# B&R Automation Studio project 8238 (part 4)

```iecst
(*** RAIL DEST MAPPING FOR RAIL DESTINATIONS ***)

DEST_SIZE := rail_destination_1;
DEST_RAIL := 0;
DEST_NUM := 0;
IF DEST_SIZE > 0 THEN
	FOR DEST_INDEX := 1 TO DEST_SIZE DO
		CASE DEST_INDEX OF
		1:	DEST_RAIL := rail_destination_2; DEST_NUM := rail_destination_3;
		2:	DEST_RAIL := rail_destination_4; DEST_NUM := rail_destination_5;
		3:	DEST_RAIL := rail_destination_6; DEST_NUM := rail_destination_7;
		4:	DEST_RAIL := rail_destination_8; DEST_NUM := rail_destination_9;
		5:	DEST_RAIL := rail_destination_10; DEST_NUM := rail_destination_11;
		6:	DEST_RAIL := rail_destination_12; DEST_NUM := rail_destination_13;
		7:	DEST_RAIL := rail_destination_14; DEST_NUM := rail_destination_15;
		8:	DEST_RAIL := rail_destination_16; DEST_NUM := rail_destination_17;
		9:	DEST_RAIL := rail_destination_18; DEST_NUM := rail_destination_19;
		10:	DEST_RAIL := rail_destination_20; DEST_NUM := rail_destination_21;
		11:	DEST_RAIL := rail_destination_22; DEST_NUM := rail_destination_23;
		12:	DEST_RAIL := rail_destination_24; DEST_NUM := rail_destination_25;
		13:	DEST_RAIL := rail_destination_26; DEST_NUM := rail_destination_27;
		14:	DEST_RAIL := rail_destination_28; DEST_NUM := rail_destination_29;
		15:	DEST_RAIL := rail_destination_30; DEST_NUM := rail_destination_31;
		16:	DEST_RAIL := rail_destination_32; DEST_NUM := rail_destination_33;
		17:	DEST_RAIL := rail_destination_34; DEST_NUM := rail_destination_35;
		18:	DEST_RAIL := rail_destination_36; DEST_NUM := rail_destination_37;
		19:	DEST_RAIL := rail_destination_38; DEST_NUM := rail_destination_39;
		20:	DEST_RAIL := rail_destination_40; DEST_NUM := rail_destination_41;
		21:	DEST_RAIL := rail_destination_42; DEST_NUM := rail_destination_43;
		22:	DEST_RAIL := rail_destination_44; DEST_NUM := rail_destination_45;
		23:	DEST_RAIL := rail_destination_46; DEST_NUM := rail_destination_47;
		24:	DEST_RAIL := rail_destination_48; DEST_NUM := rail_destination_49;
		25:	DEST_RAIL := rail_destination_50; DEST_NUM := rail_destination_51;
		26:	DEST_RAIL := rail_destination_52; DEST_NUM := rail_destination_53;
		27:	DEST_RAIL := rail_destination_54; DEST_NUM := rail_destination_55;
		28:	DEST_RAIL := rail_destination_56; DEST_NUM := rail_destination_57;
		29:	DEST_RAIL := rail_destination_58; DEST_NUM := rail_destination_59;
		30:	DEST_RAIL := rail_destination_60; DEST_NUM := rail_destination_61;
		31:	DEST_RAIL := rail_destination_62; DEST_NUM := rail_destination_63;
		32:	DEST_RAIL := rail_destination_64; DEST_NUM := rail_destination_65;
		33:	DEST_RAIL := rail_destination_66; DEST_NUM := rail_destination_67;
		34:	DEST_RAIL := rail_destination_68; DEST_NUM := rail_destination_69;
		35:	DEST_RAIL := rail_destination_70; DEST_NUM := rail_destination_71;
		36:	DEST_RAIL := rail_destination_72; DEST_NUM := rail_destination_73;
		37:	DEST_RAIL := rail_destination_74; DEST_NUM := rail_destination_75;
		38:	DEST_RAIL := rail_destination_76; DEST_NUM := rail_destination_77;
		39:	DEST_RAIL := rail_destination_78; DEST_NUM := rail_destination_79;
		40:	DEST_RAIL := rail_destination_80; DEST_NUM := rail_destination_81;
		41:	DEST_RAIL := rail_destination_82; DEST_NUM := rail_destination_83;
		42:	DEST_RAIL := rail_destination_84; DEST_NUM := rail_destination_85;
		43:	DEST_RAIL := rail_destination_86; DEST_NUM := rail_destination_87;
		44:	DEST_RAIL := rail_destination_88; DEST_NUM := rail_destination_89;
		45:	DEST_RAIL := rail_destination_90; DEST_NUM := rail_destination_91;
		46:	DEST_RAIL := rail_destination_92; DEST_NUM := rail_destination_93;
		47:	DEST_RAIL := rail_destination_94; DEST_NUM := rail_destination_95;
		48:	DEST_RAIL := rail_destination_96; DEST_NUM := rail_destination_97;
		49:	DEST_RAIL := rail_destination_98; DEST_NUM := rail_destination_99;
		50:	DEST_RAIL := rail_destination_100; DEST_NUM := rail_destination_101;
		END_CASE;
		CASE DEST_RAIL OF
		1:	r1.destination := DEST_NUM;
		2:	r2.destination := DEST_NUM;
		3:	r3.destination := DEST_NUM;
		4:	r4.destination := DEST_NUM;
		5:	r5.destination := DEST_NUM;
		6:	r6.destination := DEST_NUM;
		7:	r7.destination := DEST_NUM;
		8:	r8.destination := DEST_NUM;
		9:	r9.destination := DEST_NUM;
		10:	r10.destination := DEST_NUM;
		11:	r11.destination := DEST_NUM;
		12:	r12.destination := DEST_NUM;
		13:	r13.destination := DEST_NUM;
		14:	r14.destination := DEST_NUM;
		15:	r15.destination := DEST_NUM;
		16:	r16.destination := DEST_NUM;
		17:	r17.destination := DEST_NUM;
		18:	r18.destination := DEST_NUM;
		19:	r19.destination := DEST_NUM;
		20:	r20.destination := DEST_NUM;
		21:	r21.destination := DEST_NUM;
		22:	r22.destination := DEST_NUM;
		23:	r23.destination := DEST_NUM;
		24:	r24.destination := DEST_NUM;
		25:	r25.destination := DEST_NUM;
		26:	r26.destination := DEST_NUM;
		27:	r27.destination := DEST_NUM;
		28:	r28.destination := DEST_NUM;
		29:	r29.destination := DEST_NUM;
		30:	r30.destination := DEST_NUM;
		31:	r31.destination := DEST_NUM;
		32:	r32.destination := DEST_NUM;
		33:	r33.destination := DEST_NUM;
		34:	r34.destination := DEST_NUM;
		35:	r35.destination := DEST_NUM;
		36:	r36.destination := DEST_NUM;
		37:	r37.destination := DEST_NUM;
		38:	r38.destination := DEST_NUM;
		39:	r39.destination := DEST_NUM;
		40:	r40.destination := DEST_NUM;
		41:	r41.destination := DEST_NUM;
		42:	r42.destination := DEST_NUM;
		43:	r43.destination := DEST_NUM;
		44:	r44.destination := DEST_NUM;
		45:	r45.destination := DEST_NUM;
		46:	r46.destination := DEST_NUM;
		47:	r47.destination := DEST_NUM;
		48:	r48.destination := DEST_NUM;
		49:	r49.destination := DEST_NUM;
		50:	r50.destination := DEST_NUM;
		51:	r51.destination := DEST_NUM;
		52:	r52.destination := DEST_NUM;
		53:	r53.destination := DEST_NUM;
		54:	r54.destination := DEST_NUM;
		55:	r55.destination := DEST_NUM;
		56:	r56.destination := DEST_NUM;
		57:	r57.destination := DEST_NUM;
		58:	r58.destination := DEST_NUM;
		59:	r59.destination := DEST_NUM;
		60:	r60.destination := DEST_NUM;
		61:	r61.destination := DEST_NUM;
		62:	r62.destination := DEST_NUM;
		63:	r63.destination := DEST_NUM;
		64:	r64.destination := DEST_NUM;
		65:	r65.destination := DEST_NUM;
		66:	r66.destination := DEST_NUM;
		67:	r67.destination := DEST_NUM;
		68:	r68.destination := DEST_NUM;
		69:	r69.destination := DEST_NUM;
		70:	r70.destination := DEST_NUM;
		71:	r71.destination := DEST_NUM;
		72:	r72.destination := DEST_NUM;
		73:	r73.destination := DEST_NUM;
		74:	r74.destination := DEST_NUM;
		END_CASE;
	END_FOR;
END_IF;
rail_destination_1 := 0;
rail_destination_2 := 0;
rail_destination_3 := 0;
rail_destination_4 := 0;
rail_destination_5 := 0;
rail_destination_6 := 0;
rail_destination_7 := 0;
rail_destination_8 := 0;
rail_destination_9 := 0;
rail_destination_10 := 0;
rail_destination_11 := 0;
rail_destination_12 := 0;
rail_destination_13 := 0;
rail_destination_14 := 0;
rail_destination_15 := 0;
rail_destination_16 := 0;
rail_destination_17 := 0;
rail_destination_18 := 0;
rail_destination_19 := 0;
rail_destination_20 := 0;
rail_destination_21 := 0;
rail_destination_22 := 0;
rail_destination_23 := 0;
rail_destination_24 := 0;
rail_destination_25 := 0;
rail_destination_26 := 0;
rail_destination_27 := 0;
rail_destination_28 := 0;
rail_destination_29 := 0;
rail_destination_30 := 0;
rail_destination_31 := 0;
rail_destination_32 := 0;
rail_destination_33 := 0;
rail_destination_34 := 0;
rail_destination_35 := 0;
rail_destination_36 := 0;
rail_destination_37 := 0;
rail_destination_38 := 0;
rail_destination_39 := 0;
rail_destination_40 := 0;
rail_destination_41 := 0;
rail_destination_42 := 0;
rail_destination_43 := 0;
rail_destination_44 := 0;
rail_destination_45 := 0;
rail_destination_46 := 0;
rail_destination_47 := 0;
rail_destination_48 := 0;
rail_destination_49 := 0;
rail_destination_50 := 0;
rail_destination_51 := 0;
rail_destination_52 := 0;
rail_destination_53 := 0;
rail_destination_54 := 0;
rail_destination_55 := 0;
rail_destination_56 := 0;
rail_destination_57 := 0;
rail_destination_58 := 0;
rail_destination_59 := 0;
rail_destination_60 := 0;
rail_destination_61 := 0;
rail_destination_62 := 0;
rail_destination_63 := 0;
rail_destination_64 := 0;
rail_destination_65 := 0;
rail_destination_66 := 0;
rail_destination_67 := 0;
rail_destination_68 := 0;
rail_destination_69 := 0;
rail_destination_70 := 0;
rail_destination_71 := 0;
rail_destination_72 := 0;
rail_destination_73 := 0;
rail_destination_74 := 0;
rail_destination_75 := 0;
rail_destination_76 := 0;
rail_destination_77 := 0;
rail_destination_78 := 0;
rail_destination_79 := 0;
rail_destination_80 := 0;
rail_destination_81 := 0;
rail_destination_82 := 0;
rail_destination_83 := 0;
rail_destination_84 := 0;
rail_destination_85 := 0;
rail_destination_86 := 0;
rail_destination_87 := 0;
rail_destination_88 := 0;
rail_destination_89 := 0;
rail_destination_90 := 0;
rail_destination_91 := 0;
rail_destination_92 := 0;
rail_destination_93 := 0;
rail_destination_94 := 0;
rail_destination_95 := 0;
rail_destination_96 := 0;
rail_destination_97 := 0;
rail_destination_98 := 0;
rail_destination_99 := 0;
rail_destination_100 := 0;
rail_destination_101 := 0;

(*** RESET CLEARING DEST, FIRE, AND GOING_TO ***)

(*** Rail 1 ***)
IF r1.reset THEN
	r1.fire := 0;
	IF r1.destination = 61 THEN
		r61.going_to := 0;
	END_IF;
	r1.destination := 0;
END_IF;

(*** Rail 2 ***)
IF r2.reset THEN
	r2.fire := 0;
	IF r2.destination = 61 THEN
		r61.going_to := 0;
	END_IF;
	r2.destination := 0;
END_IF;

(*** Rail 3 ***)
IF r3.reset THEN
	r3.fire := 0;
	IF r3.destination = 61 THEN
		r61.going_to := 0;
	END_IF;
	r3.destination := 0;
END_IF;

(*** Rail 4 ***)
IF r4.reset THEN
	r4.fire := 0;
	IF r4.destination = 61 THEN
		r61.going_to := 0;
	END_IF;
	r4.destination := 0;
END_IF;

(*** Rail 5 ***)
IF r5.reset THEN
	r5.fire := 0;
	IF r5.destination = 61 THEN
		r61.going_to := 0;
	END_IF;
	r5.destination := 0;
END_IF;

(*** Rail 6 ***)
IF r6.reset THEN
	r6.fire := 0;
	IF r6.destination = 61 THEN
		r61.going_to := 0;
	END_IF;
	r6.destination := 0;
END_IF;

(*** Rail 7 ***)
IF r7.reset THEN
	r7.fire := 0;
	IF r7.destination = 61 THEN
		r61.going_to := 0;
	END_IF;
	r7.destination := 0;
END_IF;

(*** Rail 8 ***)
IF r8.reset THEN
	r8.fire := 0;
	IF r8.destination = 61 THEN
		r61.going_to := 0;
	END_IF;
	r8.destination := 0;
END_IF;

(*** Rail 9 ***)
IF r9.reset THEN
	r9.fire := 0;
	IF r9.destination = 61 THEN
		r61.going_to := 0;
	END_IF;
	r9.destination := 0;
END_IF;

(*** Rail 10 ***)
IF r10.reset THEN
	r10.fire := 0;
	IF r10.destination = 61 THEN
		r61.going_to := 0;
	END_IF;
	r10.destination := 0;
END_IF;

(*** Rail 11 ***)
IF r11.reset THEN
	r11.fire := 0;
	IF r11.destination = 61 THEN
		r61.going_to := 0;
	END_IF;
	r11.destination := 0;
END_IF;

(*** Rail 12 ***)
IF r12.reset THEN
	r12.fire := 0;
	IF r12.destination = 63 THEN
		r63.going_to := 0;
	END_IF;
	r12.destination := 0;
END_IF;

(*** Rail 13 ***)
IF r13.reset THEN
	r13.fire := 0;
	IF r13.destination = 63 THEN
		r63.going_to := 0;
	END_IF;
	r13.destination := 0;
END_IF;

(*** Rail 14 ***)
IF r14.reset THEN
	r14.fire := 0;
	IF r14.destination = 63 THEN
		r63.going_to := 0;
	END_IF;
	r14.destination := 0;
END_IF;

(*** Rail 15 ***)
IF r15.reset THEN
	r15.fire := 0;
	IF r15.destination = 63 THEN
		r63.going_to := 0;
	END_IF;
	r15.destination := 0;
END_IF;

(*** Rail 16 ***)
IF r16.reset THEN
	r16.fire := 0;
	IF r16.destination = 63 THEN
		r63.going_to := 0;
	END_IF;
	r16.destination := 0;
END_IF;

(*** Rail 17 ***)
IF r17.reset THEN
	r17.fire := 0;
	IF r17.destination = 63 THEN
		r63.going_to := 0;
	END_IF;
	r17.destination := 0;
END_IF;

(*** Rail 18 ***)
IF r18.reset THEN
	r18.fire := 0;
	IF r18.destination = 63 THEN
		r63.going_to := 0;
	END_IF;
	r18.destination := 0;
END_IF;

(*** Rail 19 ***)
IF r19.reset THEN
	r19.fire := 0;
	IF r19.destination = 63 THEN
		r63.going_to := 0;
	END_IF;
	r19.destination := 0;
END_IF;

(*** Rail 20 ***)
IF r20.reset THEN
	r20.fire := 0;
	IF r20.destination = 63 THEN
		r63.going_to := 0;
	END_IF;
	r20.destination := 0;
END_IF;

(*** Rail 21 ***)
IF r21.reset THEN
	r21.fire := 0;
	IF r21.destination = 63 THEN
		r63.going_to := 0;
	END_IF;
	r21.destination := 0;
END_IF;

(*** Rail 22 ***)
IF r22.reset THEN
	r22.fire := 0;
	IF r22.destination = 63 THEN
		r63.going_to := 0;
	END_IF;
	r22.destination := 0;
END_IF;

(*** Rail 23 ***)
IF r23.reset THEN
	r23.fire := 0;
	IF r23.destination = 63 THEN
		r63.going_to := 0;
	END_IF;
	r23.destination := 0;
END_IF;

(*** Rail 24 ***)
IF r24.reset THEN
	r24.fire := 0;
	IF r24.destination = 63 THEN
		r63.going_to := 0;
	END_IF;
	r24.destination := 0;
END_IF;

(*** Rail 25 ***)
IF r25.reset THEN
	r25.fire := 0;
	IF r25.destination = 63 THEN
		r63.going_to := 0;
	END_IF;
	r25.destination := 0;
END_IF;

(*** Rail 26 ***)
IF r26.reset THEN
	r26.fire := 0;
	IF r26.destination = 63 THEN
		r63.going_to := 0;
	END_IF;
	r26.destination := 0;
END_IF;

(*** Rail 27 ***)
IF r27.reset THEN
	r27.fire := 0;
	IF r27.destination = 63 THEN
		r63.going_to := 0;
	END_IF;
	r27.destination := 0;
END_IF;

(*** Rail 28 ***)
IF r28.reset THEN
	r28.fire := 0;
	IF r28.destination = 63 THEN
		r63.going_to := 0;
	END_IF;
	r28.destination := 0;
END_IF;

(*** Rail 29 ***)
IF r29.reset THEN
	r29.fire := 0;
	IF r29.destination = 63 THEN
		r63.going_to := 0;
	END_IF;
	r29.destination := 0;
END_IF;

(*** Rail 30 ***)
IF r30.reset THEN
	r30.fire := 0;
	IF r30.destination = 63 THEN
		r63.going_to := 0;
	END_IF;
	r30.destination := 0;
END_IF;

(*** Rail 31 ***)
IF r31.reset THEN
	r31.fire := 0;
	IF r31.destination = 63 THEN
		r63.going_to := 0;
	END_IF;
	r31.destination := 0;
END_IF;

(*** Rail 32 ***)
IF r32.reset THEN
	r32.fire := 0;
	IF r32.destination = 63 THEN
		r63.going_to := 0;
	END_IF;
	r32.destination := 0;
END_IF;

(*** Rail 33 ***)
IF r33.reset THEN
	r33.fire := 0;
	IF r33.destination = 63 THEN
		r63.going_to := 0;
	END_IF;
	r33.destination := 0;
END_IF;

(*** Rail 34 ***)
IF r34.reset THEN
	r34.fire := 0;
	IF r34.destination = 63 THEN
		r63.going_to := 0;
	END_IF;
	r34.destination := 0;
END_IF;

(*** Rail 35 ***)
IF r35.reset THEN
	r35.fire := 0;
	IF r35.destination = 63 THEN
		r63.going_to := 0;
	END_IF;
	r35.destination := 0;
END_IF;

(*** Rail 36 ***)
IF r36.reset THEN
	r36.fire := 0;
	IF r36.destination = 63 THEN
		r63.going_to := 0;
	END_IF;
	r36.destination := 0;
END_IF;

(*** Rail 37 ***)
IF r37.reset THEN
	r37.fire := 0;
	IF r37.destination = 66 THEN
		r66.going_to := 0;
	END_IF;
	r37.destination := 0;
END_IF;

(*** Rail 38 ***)
IF r38.reset THEN
	r38.fire := 0;
	IF r38.destination = 66 THEN
		r66.going_to := 0;
	END_IF;
	r38.destination := 0;
END_IF;

(*** Rail 39 ***)
IF r39.reset THEN
	r39.fire := 0;
	IF r39.destination = 66 THEN
		r66.going_to := 0;
	END_IF;
	r39.destination := 0;
END_IF;

(*** Rail 40 ***)
IF r40.reset THEN
	r40.fire := 0;
	IF r40.destination = 66 THEN
		r66.going_to := 0;
	END_IF;
	r40.destination := 0;
END_IF;

(*** Rail 41 ***)
IF r41.reset THEN
	r41.fire := 0;
	IF r41.destination = 66 THEN
		r66.going_to := 0;
	END_IF;
	r41.destination := 0;
END_IF;

(*** Rail 42 ***)
IF r42.reset THEN
	r42.fire := 0;
	IF r42.destination = 66 THEN
		r66.going_to := 0;
	END_IF;
	r42.destination := 0;
END_IF;

(*** Rail 43 ***)
IF r43.reset THEN
	r43.fire := 0;
	IF r43.destination = 65 THEN
		r65.going_to := 0;
	END_IF;
	r43.destination := 0;
END_IF;

(*** Rail 44 ***)
IF r44.reset THEN
	r44.fire := 0;
	IF r44.destination = 65 THEN
		r65.going_to := 0;
	END_IF;
	r44.destination := 0;
END_IF;

(*** Rail 45 ***)
IF r45.reset THEN
	r45.fire := 0;
	IF r45.destination = 65 THEN
		r65.going_to := 0;
	END_IF;
	r45.destination := 0;
END_IF;

(*** Rail 46 ***)
IF r46.reset THEN
	r46.fire := 0;
	IF r46.destination = 65 THEN
		r65.going_to := 0;
	END_IF;
	r46.destination := 0;
END_IF;

(*** Rail 47 ***)
IF r47.reset THEN
	r47.fire := 0;
	IF r47.destination = 65 THEN
		r65.going_to := 0;
	END_IF;
	r47.destination := 0;
END_IF;

(*** Rail 48 ***)
IF r48.reset THEN
	r48.fire := 0;
	IF r48.destination = 65 THEN
		r65.going_to := 0;
	END_IF;
	r48.destination := 0;
END_IF;

(*** Rail 49 ***)
IF r49.reset THEN
	r49.fire := 0;
	IF r49.destination = 69 THEN
		r69.going_to := 0;
	END_IF;
	r49.destination := 0;
END_IF;

(*** Rail 50 ***)
IF r50.reset THEN
	r50.fire := 0;
	IF r50.destination = 69 THEN
		r69.going_to := 0;
	END_IF;
	r50.destination := 0;
END_IF;

(*** Rail 51 ***)
IF r51.reset THEN
	r51.fire := 0;
	IF r51.destination = 69 THEN
		r69.going_to := 0;
	END_IF;
	r51.destination := 0;
END_IF;

(*** Rail 52 ***)
IF r52.reset THEN
	r52.fire := 0;
	IF r52.destination = 69 THEN
		r69.going_to := 0;
	END_IF;
	r52.destination := 0;
END_IF;

(*** Rail 53 ***)
IF r53.reset THEN
	r53.fire := 0;
	IF r53.destination = 69 THEN
		r69.going_to := 0;
	END_IF;
	r53.destination := 0;
END_IF;

(*** Rail 54 ***)
IF r54.reset THEN
	r54.fire := 0;
	IF r54.destination = 69 THEN
		r69.going_to := 0;
	END_IF;
	r54.destination := 0;
END_IF;

(*** Rail 55 ***)
IF r55.reset THEN
	r55.fire := 0;
	IF r55.destination = 68 THEN
		r68.going_to := 0;
	END_IF;
	r55.destination := 0;
END_IF;

(*** Rail 56 ***)
IF r56.reset THEN
	r56.fire := 0;
	IF r56.destination = 68 THEN
		r68.going_to := 0;
	END_IF;
	r56.destination := 0;
END_IF;

(*** Rail 57 ***)
IF r57.reset THEN
	r57.fire := 0;
	IF r57.destination = 68 THEN
		r68.going_to := 0;
	END_IF;
	r57.destination := 0;
END_IF;

(*** Rail 58 ***)
IF r58.reset THEN
	r58.fire := 0;
	IF r58.destination = 68 THEN
		r68.going_to := 0;
	END_IF;
	r58.destination := 0;
END_IF;

(*** Rail 59 ***)
IF r59.reset THEN
	r59.fire := 0;
	IF r59.destination = 68 THEN
		r68.going_to := 0;
	END_IF;
	r59.destination := 0;
END_IF;

(*** Rail 60 ***)
IF r60.reset THEN
	r60.fire := 0;
	IF r60.destination = 68 THEN
		r68.going_to := 0;
	END_IF;
	r60.destination := 0;
END_IF;

(*** Rail 61 ***)
IF r61.reset THEN
	r61.fire := 0;
	r61.destination := 0;
END_IF;

(*** Rail 62 ***)
IF r62.reset THEN
	r62.fire := 0;
	r62.destination := 0;
END_IF;

(*** Rail 63 ***)
IF r63.reset THEN
	r63.fire := 0;
	r63.destination := 0;
END_IF;

(*** Rail 64 ***)
IF r64.reset THEN
	r64.fire := 0;
	r64.destination := 0;
END_IF;

(*** Rail 65 ***)
IF r65.reset THEN
	r65.fire := 0;
	r65.destination := 0;
END_IF;

(*** Rail 66 ***)
IF r66.reset THEN
	r66.fire := 0;
	r66.destination := 0;
END_IF;

(*** Rail 67 ***)
IF r67.reset THEN
	r67.fire := 0;
	r67.destination := 0;
END_IF;

(*** Rail 68 ***)
IF r68.reset THEN
	r68.fire := 0;
	r68.destination := 0;
END_IF;

(*** Rail 69 ***)
IF r69.reset THEN
	r69.fire := 0;
	r69.destination := 0;
END_IF;

(*** Rail 70 ***)
IF r70.reset THEN
	r70.fire := 0;
	r70.destination := 0;
END_IF;

(*** Rail 71 ***)
IF r71.reset THEN
	r71.fire := 0;
	r71.destination := 0;
END_IF;

(*** Rail 72 ***)
IF r72.reset THEN
	r72.fire := 0;
	r72.destination := 0;
END_IF;

(*** Rail 73 ***)
IF r73.reset THEN
	r73.fire := 0;
	r73.destination := 0;
END_IF;

(*** Rail 74 ***)
IF r74.reset THEN
	r74.fire := 0;
	r74.destination := 0;
END_IF;

(*** Conveyor Stop Signals ***)

conveyor_stop_1 := conveyor_stop_word_1.0;
conveyor_stop_2 := conveyor_stop_word_1.1;
conveyor_stop_3 := conveyor_stop_word_1.2;
conveyor_stop_4 := conveyor_stop_word_1.3;

END_PROGRAM
```

### Program Logical/LIFTS (IEC, version 1.00.1)

#### LIFTS.st
```iecst
(********************************************************************
 * Program: lifts
 * File: lifts.st
 ********************************************************************)
PROGRAM _CYCLIC
END_PROGRAM
```

#### Variables.var - not listed in the package file held
```iecst
VAR
	slant_timeout : BOOL;
	test_bit_a : BOOL;
	test_bit_b : BOOL;
END_VAR
```

#### Cyclic.ld - not listed in the package file held
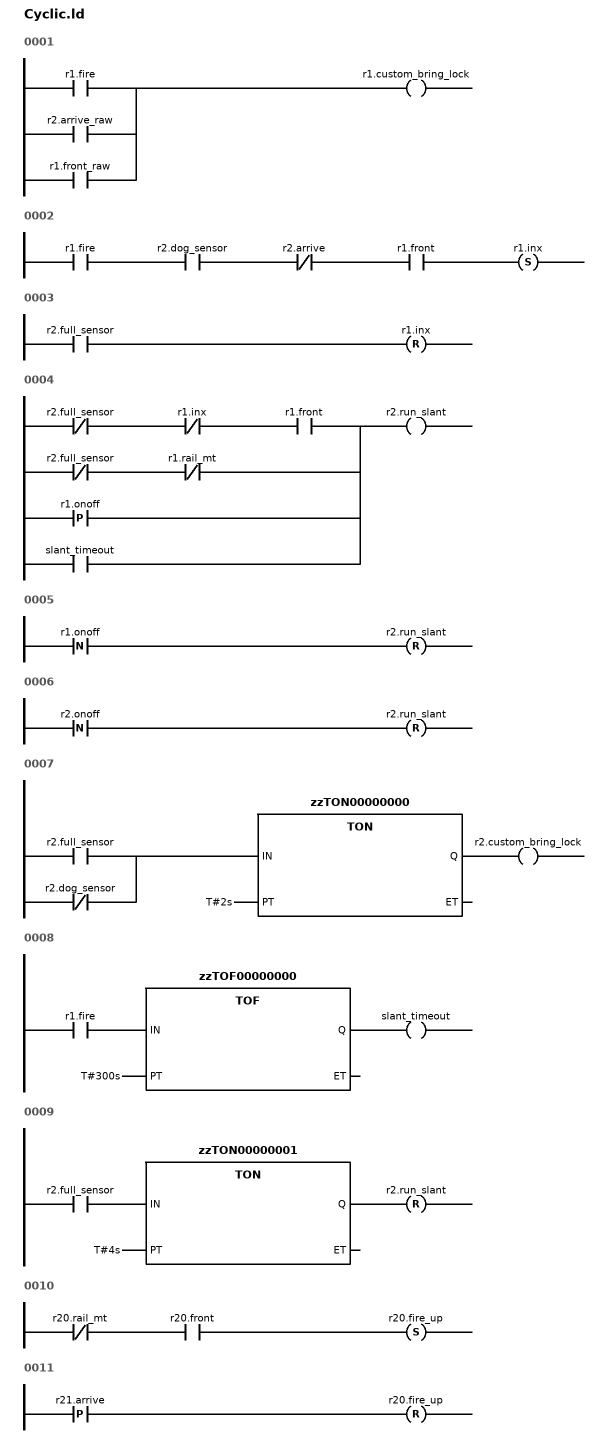
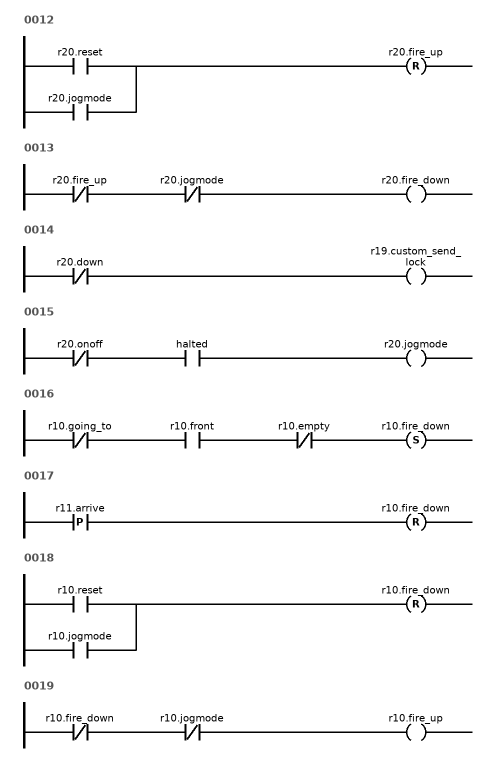
Ladder, written as Structured Text:
```iecst
PROGRAM _CYCLIC
VAR
    _e1 : R_TRIG;
    _e2 : F_TRIG;
    _e3 : F_TRIG;
    _e4 : R_TRIG;
    _e5 : R_TRIG;
END_VAR
(* Network 1 *)
r1.custom_bring_lock := r1.fire OR r2.arrive_raw OR r1.front_raw;

(* Network 2 *)
IF r1.fire AND r2.dog_sensor AND NOT r2.arrive AND r1.front THEN r1.inx := TRUE; END_IF;

(* Network 3 *)
IF r2.full_sensor THEN r1.inx := FALSE; END_IF;

(* Network 4 *)
_e1(CLK := r1.onoff);
r2.run_slant := (NOT r2.full_sensor AND ((NOT r1.inx AND r1.front) OR NOT r1.rail_mt)) OR _e1.Q OR slant_timeout;

(* Network 5 *)
_e2(CLK := r1.onoff);
IF _e2.Q THEN r2.run_slant := FALSE; END_IF;

(* Network 6 *)
_e3(CLK := r2.onoff);
IF _e3.Q THEN r2.run_slant := FALSE; END_IF;

(* Network 7 *)
zzTON00000000(IN := r2.full_sensor OR NOT r2.dog_sensor, PT := T#2s);
r2.custom_bring_lock := zzTON00000000.Q;

(* Network 8 *)
zzTOF00000000(IN := r1.fire, PT := T#300s);
slant_timeout := zzTOF00000000.Q;

(* Network 9 *)
zzTON00000001(IN := r2.full_sensor, PT := T#4s);
IF zzTON00000001.Q THEN r2.run_slant := FALSE; END_IF;

(* Network 10 *)
IF NOT r20.rail_mt AND r20.front THEN r20.fire_up := TRUE; END_IF;

(* Network 11 *)
_e4(CLK := r21.arrive);
IF _e4.Q THEN r20.fire_up := FALSE; END_IF;

(* Network 12 *)
IF r20.reset OR r20.jogmode THEN r20.fire_up := FALSE; END_IF;

(* Network 13 *)
r20.fire_down := NOT r20.fire_up AND NOT r20.jogmode;

(* Network 14 *)
r19.custom_send_lock := NOT r20.down;

(* Network 15 *)
r20.jogmode := NOT r20.onoff AND halted;

(* Network 16 *)
IF NOT r10.going_to AND r10.front AND NOT r10.empty THEN r10.fire_down := TRUE; END_IF;

(* Network 17 *)
_e5(CLK := r11.arrive);
IF _e5.Q THEN r10.fire_down := FALSE; END_IF;

(* Network 18 *)
IF r10.reset OR r10.jogmode THEN r10.fire_down := FALSE; END_IF;

(* Network 19 *)
r10.fire_up := NOT r10.fire_down AND NOT r10.jogmode;
END_PROGRAM
```

### Program Logical/RAIL_SUB (IEC, version 1.00.1) - RAIL_SUB

#### RAIL_SUB.st
```iecst
(********************************************************************
 * Program: st_rails
 * File: st_rails.st
 ********************************************************************)
PROGRAM _CYCLIC
(***	RAILS	***)
(*
  This section maps the plc state of io_ok and manages fire bits
*)

	(***	Rail: 1	***)
	IF r1.fire_ns THEN r1.destination := 0; END_IF;
	IF r1.destination = 61 THEN
		IF NOT(r61.going_to) AND NOT(r1.reset) AND NOT(r61.insert_reset) THEN
			r61.going_to := TRUE;
			r1.fire := TRUE;
		END_IF;

		IF r1.fire AND r61.insert_reset THEN
			r1.fire := FALSE;
		END_IF;
	END_IF;

	(***	Rail: 2	***)
	IF r2.fire_ns THEN r2.destination := 0; END_IF;
	IF r2.destination = 61 THEN
		IF NOT(r61.going_to) AND NOT(r2.reset) AND NOT(r61.insert_reset) THEN
			r61.going_to := TRUE;
			r2.fire := TRUE;
		END_IF;

		IF r2.fire AND r61.insert_reset THEN
			r2.fire := FALSE;
		END_IF;
	END_IF;

	(***	Rail: 3	***)
	IF r3.fire_ns THEN r3.destination := 0; END_IF;
	IF r3.destination = 61 THEN
		IF NOT(r61.going_to) AND NOT(r3.reset) AND NOT(r61.insert_reset) THEN
			r61.going_to := TRUE;
			r3.fire := TRUE;
		END_IF;

		IF r3.fire AND r61.insert_reset THEN
			r3.fire := FALSE;
		END_IF;
	END_IF;

	(***	Rail: 4	***)
	IF r4.fire_ns THEN r4.destination := 0; END_IF;
	IF r4.destination = 61 THEN
		IF NOT(r61.going_to) AND NOT(r4.reset) AND NOT(r61.insert_reset) THEN
			r61.going_to := TRUE;
			r4.fire := TRUE;
		END_IF;

		IF r4.fire AND r61.insert_reset THEN
			r4.fire := FALSE;
		END_IF;
	END_IF;

	(***	Rail: 5	***)
	IF r5.fire_ns THEN r5.destination := 0; END_IF;
	IF r5.destination = 61 THEN
		IF NOT(r61.going_to) AND NOT(r5.reset) AND NOT(r61.insert_reset) THEN
			r61.going_to := TRUE;
			r5.fire := TRUE;
		END_IF;

		IF r5.fire AND r61.insert_reset THEN
			r5.fire := FALSE;
		END_IF;
	END_IF;

	(***	Rail: 6	***)
	IF r6.fire_ns THEN r6.destination := 0; END_IF;
	IF r6.destination = 61 THEN
		IF NOT(r61.going_to) AND NOT(r6.reset) AND NOT(r61.insert_reset) THEN
			r61.going_to := TRUE;
			r6.fire := TRUE;
		END_IF;

		IF r6.fire AND r61.insert_reset THEN
			r6.fire := FALSE;
		END_IF;
	END_IF;

	(***	Rail: 7	***)
	IF r7.fire_ns THEN r7.destination := 0; END_IF;
	IF r7.destination = 61 THEN
		IF NOT(r61.going_to) AND NOT(r7.reset) AND NOT(r61.insert_reset) THEN
			r61.going_to := TRUE;
			r7.fire := TRUE;
		END_IF;

		IF r7.fire AND r61.insert_reset THEN
			r7.fire := FALSE;
		END_IF;
	END_IF;

	(***	Rail: 8	***)
	IF r8.fire_ns THEN r8.destination := 0; END_IF;
	IF r8.destination = 61 THEN
		IF NOT(r61.going_to) AND NOT(r8.reset) AND NOT(r61.insert_reset) THEN
			r61.going_to := TRUE;
			r8.fire := TRUE;
		END_IF;

		IF r8.fire AND r61.insert_reset THEN
			r8.fire := FALSE;
		END_IF;
	END_IF;

	(***	Rail: 9	***)
	IF r9.fire_ns THEN r9.destination := 0; END_IF;
	IF r9.destination = 61 THEN
		IF NOT(r61.going_to) AND NOT(r9.reset) AND NOT(r61.insert_reset) THEN
			r61.going_to := TRUE;
			r9.fire := TRUE;
		END_IF;

		IF r9.fire AND r61.insert_reset THEN
			r9.fire := FALSE;
		END_IF;
	END_IF;

	(***	Rail: 10	***)
	IF r10.fire_ns THEN r10.destination := 0; END_IF;
	IF r10.destination = 61 THEN
		IF NOT(r61.going_to) AND NOT(r10.reset) AND NOT(r61.insert_reset) THEN
			r61.going_to := TRUE;
			r10.fire := TRUE;
		END_IF;

		IF r10.fire AND r61.insert_reset THEN
			r10.fire := FALSE;
		END_IF;
	END_IF;

	(***	Rail: 11	***)
	IF r11.fire_ns THEN r11.destination := 0; END_IF;
	IF r11.destination = 61 THEN
		IF NOT(r61.going_to) AND NOT(r11.reset) AND NOT(r61.insert_reset) THEN
			r61.going_to := TRUE;
			r11.fire := TRUE;
		END_IF;

		IF r11.fire AND r61.insert_reset THEN
			r11.fire := FALSE;
		END_IF;
	END_IF;

	(***	Rail: 12	***)
	IF r12.fire_ns THEN r12.destination := 0; END_IF;
	IF r12.destination = 63 THEN
		IF NOT(r63.going_to) AND NOT(r12.reset) AND NOT(r63.insert_reset) THEN
			r63.going_to := TRUE;
			r12.fire := TRUE;
		END_IF;

		IF r12.fire AND r63.insert_reset THEN
			r12.fire := FALSE;
		END_IF;
	END_IF;

	(***	Rail: 13	***)
	IF r13.fire_ns THEN r13.destination := 0; END_IF;
	IF r13.destination = 63 THEN
		IF NOT(r63.going_to) AND NOT(r13.reset) AND NOT(r63.insert_reset) THEN
			r63.going_to := TRUE;
			r13.fire := TRUE;
		END_IF;

		IF r13.fire AND r63.insert_reset THEN
			r13.fire := FALSE;
		END_IF;
	END_IF;

	(***	Rail: 14	***)
	IF r14.fire_ns THEN r14.destination := 0; END_IF;
	IF r14.destination = 63 THEN
		IF NOT(r63.going_to) AND NOT(r14.reset) AND NOT(r63.insert_reset) THEN
			r63.going_to := TRUE;
			r14.fire := TRUE;
		END_IF;

		IF r14.fire AND r63.insert_reset THEN
			r14.fire := FALSE;
		END_IF;
	END_IF;

	(***	Rail: 15	***)
	IF r15.fire_ns THEN r15.destination := 0; END_IF;
	IF r15.destination = 63 THEN
		IF NOT(r63.going_to) AND NOT(r15.reset) AND NOT(r63.insert_reset) THEN
			r63.going_to := TRUE;
			r15.fire := TRUE;
		END_IF;

		IF r15.fire AND r63.insert_reset THEN
			r15.fire := FALSE;
		END_IF;
	END_IF;

	(***	Rail: 16	***)
	IF r16.fire_ns THEN r16.destination := 0; END_IF;
	IF r16.destination = 63 THEN
		IF NOT(r63.going_to) AND NOT(r16.reset) AND NOT(r63.insert_reset) THEN
			r63.going_to := TRUE;
			r16.fire := TRUE;
		END_IF;

		IF r16.fire AND r63.insert_reset THEN
			r16.fire := FALSE;
		END_IF;
	END_IF;

	(***	Rail: 17	***)
	IF r17.fire_ns THEN r17.destination := 0; END_IF;
	IF r17.destination = 63 THEN
		IF NOT(r63.going_to) AND NOT(r17.reset) AND NOT(r63.insert_reset) THEN
			r63.going_to := TRUE;
			r17.fire := TRUE;
		END_IF;

		IF r17.fire AND r63.insert_reset THEN
			r17.fire := FALSE;
		END_IF;
	END_IF;

	(***	Rail: 18	***)
	IF r18.fire_ns THEN r18.destination := 0; END_IF;
	IF r18.destination = 63 THEN
		IF NOT(r63.going_to) AND NOT(r18.reset) AND NOT(r63.insert_reset) THEN
			r63.going_to := TRUE;
			r18.fire := TRUE;
		END_IF;

		IF r18.fire AND r63.insert_reset THEN
			r18.fire := FALSE;
		END_IF;
	END_IF;

	(***	Rail: 19	***)
	IF r19.fire_ns THEN r19.destination := 0; END_IF;
	IF r19.destination = 63 THEN
		IF NOT(r63.going_to) AND NOT(r19.reset) AND NOT(r63.insert_reset) THEN
			r63.going_to := TRUE;
			r19.fire := TRUE;
		END_IF;

		IF r19.fire AND r63.insert_reset THEN
			r19.fire := FALSE;
		END_IF;
	END_IF;

	(***	Rail: 20	***)
	IF r20.fire_ns THEN r20.destination := 0; END_IF;
	IF r20.destination = 63 THEN
		IF NOT(r63.going_to) AND NOT(r20.reset) AND NOT(r63.insert_reset) THEN
			r63.going_to := TRUE;
			r20.fire := TRUE;
		END_IF;

		IF r20.fire AND r63.insert_reset THEN
			r20.fire := FALSE;
		END_IF;
	END_IF;

	(***	Rail: 21	***)
	IF r21.fire_ns THEN r21.destination := 0; END_IF;
	IF r21.destination = 63 THEN
		IF NOT(r63.going_to) AND NOT(r21.reset) AND NOT(r63.insert_reset) THEN
			r63.going_to := TRUE;
			r21.fire := TRUE;
		END_IF;

		IF r21.fire AND r63.insert_reset THEN
			r21.fire := FALSE;
		END_IF;
	END_IF;

	(***	Rail: 22	***)
	IF r22.fire_ns THEN r22.destination := 0; END_IF;
	IF r22.destination = 63 THEN
		IF NOT(r63.going_to) AND NOT(r22.reset) AND NOT(r63.insert_reset) THEN
			r63.going_to := TRUE;
			r22.fire := TRUE;
		END_IF;

		IF r22.fire AND r63.insert_reset THEN
			r22.fire := FALSE;
		END_IF;
	END_IF;

	(***	Rail: 23	***)
	IF r23.fire_ns THEN r23.destination := 0; END_IF;
	IF r23.destination = 63 THEN
		IF NOT(r63.going_to) AND NOT(r23.reset) AND NOT(r63.insert_reset) THEN
			r63.going_to := TRUE;
			r23.fire := TRUE;
		END_IF;

		IF r23.fire AND r63.insert_reset THEN
			r23.fire := FALSE;
		END_IF;
	END_IF;

	(***	Rail: 24	***)
	IF r24.fire_ns THEN r24.destination := 0; END_IF;
	IF r24.destination = 63 THEN
		IF NOT(r63.going_to) AND NOT(r24.reset) AND NOT(r63.insert_reset) THEN
			r63.going_to := TRUE;
			r24.fire := TRUE;
		END_IF;

		IF r24.fire AND r63.insert_reset THEN
			r24.fire := FALSE;
		END_IF;
	END_IF;

	(***	Rail: 25	***)
	IF r25.fire_ns THEN r25.destination := 0; END_IF;
	IF r25.destination = 63 THEN
		IF NOT(r63.going_to) AND NOT(r25.reset) AND NOT(r63.insert_reset) THEN
			r63.going_to := TRUE;
			r25.fire := TRUE;
		END_IF;

		IF r25.fire AND r63.insert_reset THEN
			r25.fire := FALSE;
		END_IF;
	END_IF;

	(***	Rail: 26	***)
	IF r26.fire_ns THEN r26.destination := 0; END_IF;
	IF r26.destination = 63 THEN
		IF NOT(r63.going_to) AND NOT(r26.reset) AND NOT(r63.insert_reset) THEN
			r63.going_to := TRUE;
			r26.fire := TRUE;
		END_IF;

		IF r26.fire AND r63.insert_reset THEN
			r26.fire := FALSE;
		END_IF;
	END_IF;

	(***	Rail: 27	***)
	IF r27.fire_ns THEN r27.destination := 0; END_IF;
	IF r27.destination = 63 THEN
		IF NOT(r63.going_to) AND NOT(r27.reset) AND NOT(r63.insert_reset) THEN
			r63.going_to := TRUE;
			r27.fire := TRUE;
		END_IF;

		IF r27.fire AND r63.insert_reset THEN
			r27.fire := FALSE;
		END_IF;
	END_IF;

	(***	Rail: 28	***)
	IF r28.fire_ns THEN r28.destination := 0; END_IF;
	IF r28.destination = 63 THEN
		IF NOT(r63.going_to) AND NOT(r28.reset) AND NOT(r63.insert_reset) THEN
			r63.going_to := TRUE;
			r28.fire := TRUE;
		END_IF;

		IF r28.fire AND r63.insert_reset THEN
			r28.fire := FALSE;
		END_IF;
	END_IF;

	(***	Rail: 29	***)
	IF r29.fire_ns THEN r29.destination := 0; END_IF;
	IF r29.destination = 63 THEN
		IF NOT(r63.going_to) AND NOT(r29.reset) AND NOT(r63.insert_reset) THEN
			r63.going_to := TRUE;
			r29.fire := TRUE;
		END_IF;

		IF r29.fire AND r63.insert_reset THEN
			r29.fire := FALSE;
		END_IF;
	END_IF;

	(***	Rail: 30	***)
	IF r30.fire_ns THEN r30.destination := 0; END_IF;
	IF r30.destination = 63 THEN
		IF NOT(r63.going_to) AND NOT(r30.reset) AND NOT(r63.insert_reset) THEN
			r63.going_to := TRUE;
			r30.fire := TRUE;
		END_IF;

		IF r30.fire AND r63.insert_reset THEN
			r30.fire := FALSE;
		END_IF;
	END_IF;

	(***	Rail: 31	***)
	IF r31.fire_ns THEN r31.destination := 0; END_IF;
	IF r31.destination = 63 THEN
		IF NOT(r63.going_to) AND NOT(r31.reset) AND NOT(r63.insert_reset) THEN
			r63.going_to := TRUE;
			r31.fire := TRUE;
		END_IF;

		IF r31.fire AND r63.insert_reset THEN
			r31.fire := FALSE;
		END_IF;
	END_IF;

	(***	Rail: 32	***)
	IF r32.fire_ns THEN r32.destination := 0; END_IF;
	IF r32.destination = 63 THEN
		IF NOT(r63.going_to) AND NOT(r32.reset) AND NOT(r63.insert_reset) THEN
			r63.going_to := TRUE;
			r32.fire := TRUE;
		END_IF;

		IF r32.fire AND r63.insert_reset THEN
			r32.fire := FALSE;
		END_IF;
	END_IF;

	(***	Rail: 33	***)
	IF r33.fire_ns THEN r33.destination := 0; END_IF;
	IF r33.destination = 63 THEN
		IF NOT(r63.going_to) AND NOT(r33.reset) AND NOT(r63.insert_reset) THEN
			r63.going_to := TRUE;
			r33.fire := TRUE;
		END_IF;

		IF r33.fire AND r63.insert_reset THEN
			r33.fire := FALSE;
		END_IF;
	END_IF;

	(***	Rail: 34	***)
	IF r34.fire_ns THEN r34.destination := 0; END_IF;
	IF r34.destination = 63 THEN
		IF NOT(r63.going_to) AND NOT(r34.reset) AND NOT(r63.insert_reset) THEN
			r63.going_to := TRUE;
			r34.fire := TRUE;
		END_IF;

		IF r34.fire AND r63.insert_reset THEN
			r34.fire := FALSE;
		END_IF;
	END_IF;

	(***	Rail: 35	***)
	IF r35.fire_ns THEN r35.destination := 0; END_IF;
	IF r35.destination = 63 THEN
		IF NOT(r63.going_to) AND NOT(r35.reset) AND NOT(r63.insert_reset) THEN
			r63.going_to := TRUE;
			r35.fire := TRUE;
		END_IF;

		IF r35.fire AND r63.insert_reset THEN
			r35.fire := FALSE;
		END_IF;
	END_IF;

	(***	Rail: 36	***)
	IF r36.fire_ns THEN r36.destination := 0; END_IF;
	IF r36.destination = 63 THEN
		IF NOT(r63.going_to) AND NOT(r36.reset) AND NOT(r63.insert_reset) THEN
			r63.going_to := TRUE;
			r36.fire := TRUE;
		END_IF;

		IF r36.fire AND r63.insert_reset THEN
			r36.fire := FALSE;
		END_IF;
	END_IF;

	(***	Rail: 37	***)
	IF r37.fire_ns THEN r37.destination := 0; END_IF;
	IF r37.destination = 66 THEN
		IF NOT(r66.going_to) AND NOT(r37.reset) AND NOT(r66.insert_reset) THEN
			r66.going_to := TRUE;
			r37.fire := TRUE;
		END_IF;

		IF r37.fire AND r66.insert_reset THEN
			r37.fire := FALSE;
		END_IF;
	END_IF;

	(***	Rail: 38	***)
	IF r38.fire_ns THEN r38.destination := 0; END_IF;
	IF r38.destination = 66 THEN
		IF NOT(r66.going_to) AND NOT(r38.reset) AND NOT(r66.insert_reset) THEN
			r66.going_to := TRUE;
			r38.fire := TRUE;
		END_IF;

		IF r38.fire AND r66.insert_reset THEN
			r38.fire := FALSE;
		END_IF;
	END_IF;

	(***	Rail: 39	***)
	IF r39.fire_ns THEN r39.destination := 0; END_IF;
	IF r39.destination = 66 THEN
		IF NOT(r66.going_to) AND NOT(r39.reset) AND NOT(r66.insert_reset) THEN
			r66.going_to := TRUE;
			r39.fire := TRUE;
		END_IF;

		IF r39.fire AND r66.insert_reset THEN
			r39.fire := FALSE;
		END_IF;
	END_IF;

	(***	Rail: 40	***)
	IF r40.fire_ns THEN r40.destination := 0; END_IF;
	IF r40.destination = 66 THEN
		IF NOT(r66.going_to) AND NOT(r40.reset) AND NOT(r66.insert_reset) THEN
			r66.going_to := TRUE;
			r40.fire := TRUE;
		END_IF;

		IF r40.fire AND r66.insert_reset THEN
			r40.fire := FALSE;
		END_IF;
	END_IF;

	(***	Rail: 41	***)
	IF r41.fire_ns THEN r41.destination := 0; END_IF;
	IF r41.destination = 66 THEN
		IF NOT(r66.going_to) AND NOT(r41.reset) AND NOT(r66.insert_reset) THEN
			r66.going_to := TRUE;
			r41.fire := TRUE;
		END_IF;

		IF r41.fire AND r66.insert_reset THEN
			r41.fire := FALSE;
		END_IF;
	END_IF;

	(***	Rail: 42	***)
	IF r42.fire_ns THEN r42.destination := 0; END_IF;
	IF r42.destination = 66 THEN
		IF NOT(r66.going_to) AND NOT(r42.reset) AND NOT(r66.insert_reset) THEN
			r66.going_to := TRUE;
			r42.fire := TRUE;
		END_IF;

		IF r42.fire AND r66.insert_reset THEN
			r42.fire := FALSE;
		END_IF;
	END_IF;

	(***	Rail: 43	***)
	IF r43.fire_ns THEN r43.destination := 0; END_IF;
	IF r43.destination = 65 THEN
		IF NOT(r65.going_to) AND NOT(r43.reset) AND NOT(r65.insert_reset) THEN
			r65.going_to := TRUE;
			r43.fire := TRUE;
		END_IF;

		IF r43.fire AND r65.insert_reset THEN
			r43.fire := FALSE;
		END_IF;
	END_IF;

	(***	Rail: 44	***)
	IF r44.fire_ns THEN r44.destination := 0; END_IF;
	IF r44.destination = 65 THEN
		IF NOT(r65.going_to) AND NOT(r44.reset) AND NOT(r65.insert_reset) THEN
			r65.going_to := TRUE;
			r44.fire := TRUE;
		END_IF;

		IF r44.fire AND r65.insert_reset THEN
			r44.fire := FALSE;
		END_IF;
	END_IF;

	(***	Rail: 45	***)
	IF r45.fire_ns THEN r45.destination := 0; END_IF;
	IF r45.destination = 65 THEN
		IF NOT(r65.going_to) AND NOT(r45.reset) AND NOT(r65.insert_reset) THEN
			r65.going_to := TRUE;
			r45.fire := TRUE;
		END_IF;

		IF r45.fire AND r65.insert_reset THEN
			r45.fire := FALSE;
		END_IF;
	END_IF;

	(***	Rail: 46	***)
	IF r46.fire_ns THEN r46.destination := 0; END_IF;
	IF r46.destination = 65 THEN
		IF NOT(r65.going_to) AND NOT(r46.reset) AND NOT(r65.insert_reset) THEN
			r65.going_to := TRUE;
			r46.fire := TRUE;
		END_IF;

		IF r46.fire AND r65.insert_reset THEN
			r46.fire := FALSE;
		END_IF;
	END_IF;

	(***	Rail: 47	***)
	IF r47.fire_ns THEN r47.destination := 0; END_IF;
	IF r47.destination = 65 THEN
		IF NOT(r65.going_to) AND NOT(r47.reset) AND NOT(r65.insert_reset) THEN
			r65.going_to := TRUE;
			r47.fire := TRUE;
		END_IF;

		IF r47.fire AND r65.insert_reset THEN
			r47.fire := FALSE;
		END_IF;
	END_IF;

	(***	Rail: 48	***)
	IF r48.fire_ns THEN r48.destination := 0; END_IF;
	IF r48.destination = 65 THEN
		IF NOT(r65.going_to) AND NOT(r48.reset) AND NOT(r65.insert_reset) THEN
			r65.going_to := TRUE;
			r48.fire := TRUE;
		END_IF;

		IF r48.fire AND r65.insert_reset THEN
			r48.fire := FALSE;
		END_IF;
	END_IF;

	(***	Rail: 49	***)
	IF r49.fire_ns THEN r49.destination := 0; END_IF;
	IF r49.destination = 69 THEN
		IF NOT(r69.going_to) AND NOT(r49.reset) AND NOT(r69.insert_reset) THEN
			r69.going_to := TRUE;
			r49.fire := TRUE;
		END_IF;

		IF r49.fire AND r69.insert_reset THEN
			r49.fire := FALSE;
		END_IF;
	END_IF;

	(***	Rail: 50	***)
	IF r50.fire_ns THEN r50.destination := 0; END_IF;
	IF r50.destination = 69 THEN
		IF NOT(r69.going_to) AND NOT(r50.reset) AND NOT(r69.insert_reset) THEN
			r69.going_to := TRUE;
			r50.fire := TRUE;
		END_IF;

		IF r50.fire AND r69.insert_reset THEN
			r50.fire := FALSE;
		END_IF;
	END_IF;

	(***	Rail: 51	***)
	IF r51.fire_ns THEN r51.destination := 0; END_IF;
	IF r51.destination = 69 THEN
		IF NOT(r69.going_to) AND NOT(r51.reset) AND NOT(r69.insert_reset) THEN
			r69.going_to := TRUE;
			r51.fire := TRUE;
		END_IF;

		IF r51.fire AND r69.insert_reset THEN
			r51.fire := FALSE;
		END_IF;
	END_IF;

	(***	Rail: 52	***)
	IF r52.fire_ns THEN r52.destination := 0; END_IF;
	IF r52.destination = 69 THEN
		IF NOT(r69.going_to) AND NOT(r52.reset) AND NOT(r69.insert_reset) THEN
			r69.going_to := TRUE;
			r52.fire := TRUE;
		END_IF;

		IF r52.fire AND r69.insert_reset THEN
			r52.fire := FALSE;
		END_IF;
	END_IF;

	(***	Rail: 53	***)
	IF r53.fire_ns THEN r53.destination := 0; END_IF;
	IF r53.destination = 69 THEN
		IF NOT(r69.going_to) AND NOT(r53.reset) AND NOT(r69.insert_reset) THEN
			r69.going_to := TRUE;
			r53.fire := TRUE;
		END_IF;

		IF r53.fire AND r69.insert_reset THEN
			r53.fire := FALSE;
		END_IF;
	END_IF;

	(***	Rail: 54	***)
	IF r54.fire_ns THEN r54.destination := 0; END_IF;
	IF r54.destination = 69 THEN
		IF NOT(r69.going_to) AND NOT(r54.reset) AND NOT(r69.insert_reset) THEN
			r69.going_to := TRUE;
			r54.fire := TRUE;
		END_IF;

		IF r54.fire AND r69.insert_reset THEN
			r54.fire := FALSE;
		END_IF;
	END_IF;

	(***	Rail: 55	***)
	IF r55.fire_ns THEN r55.destination := 0; END_IF;
	IF r55.destination = 68 THEN
		IF NOT(r68.going_to) AND NOT(r55.reset) AND NOT(r68.insert_reset) THEN
			r68.going_to := TRUE;
			r55.fire := TRUE;
		END_IF;

		IF r55.fire AND r68.insert_reset THEN
			r55.fire := FALSE;
		END_IF;
	END_IF;

	(***	Rail: 56	***)
	IF r56.fire_ns THEN r56.destination := 0; END_IF;
	IF r56.destination = 68 THEN
		IF NOT(r68.going_to) AND NOT(r56.reset) AND NOT(r68.insert_reset) THEN
			r68.going_to := TRUE;
			r56.fire := TRUE;
		END_IF;

		IF r56.fire AND r68.insert_reset THEN
			r56.fire := FALSE;
		END_IF;
	END_IF;

	(***	Rail: 57	***)
	IF r57.fire_ns THEN r57.destination := 0; END_IF;
	IF r57.destination = 68 THEN
		IF NOT(r68.going_to) AND NOT(r57.reset) AND NOT(r68.insert_reset) THEN
			r68.going_to := TRUE;
			r57.fire := TRUE;
		END_IF;

		IF r57.fire AND r68.insert_reset THEN
			r57.fire := FALSE;
		END_IF;
	END_IF;

	(***	Rail: 58	***)
	IF r58.fire_ns THEN r58.destination := 0; END_IF;
	IF r58.destination = 68 THEN
		IF NOT(r68.going_to) AND NOT(r58.reset) AND NOT(r68.insert_reset) THEN
			r68.going_to := TRUE;
			r58.fire := TRUE;
		END_IF;

		IF r58.fire AND r68.insert_reset THEN
			r58.fire := FALSE;
		END_IF;
	END_IF;

	(***	Rail: 59	***)
	IF r59.fire_ns THEN r59.destination := 0; END_IF;
	IF r59.destination = 68 THEN
		IF NOT(r68.going_to) AND NOT(r59.reset) AND NOT(r68.insert_reset) THEN
			r68.going_to := TRUE;
			r59.fire := TRUE;
		END_IF;

		IF r59.fire AND r68.insert_reset THEN
			r59.fire := FALSE;
		END_IF;
	END_IF;

	(***	Rail: 60	***)
	IF r60.fire_ns THEN r60.destination := 0; END_IF;
	IF r60.destination = 68 THEN
		IF NOT(r68.going_to) AND NOT(r60.reset) AND NOT(r68.insert_reset) THEN
			r68.going_to := TRUE;
			r60.fire := TRUE;
		END_IF;

		IF r60.fire AND r68.insert_reset THEN
			r60.fire := FALSE;
		END_IF;
	END_IF;

	r1.fire_r_trig(CLK:=r1.fire);
	r1.fire_f_trig(CLK:=r1.fire);
	r1.fire_os := r1.fire_r_trig.Q;
	r1.fire_ns := r1.fire_f_trig.Q;
	r1.going_to_r_trig(CLK:=r1.going_to);
	r1.going_to_f_trig(CLK:=r1.going_to);
	r1.going_to_os := r1.going_to_r_trig.Q;
	r1.going_to_ns := r1.going_to_f_trig.Q;

	r2.fire_r_trig(CLK:=r2.fire);
	r2.fire_f_trig(CLK:=r2.fire);
	r2.fire_os := r2.fire_r_trig.Q;
	r2.fire_ns := r2.fire_f_trig.Q;
	r2.going_to_r_trig(CLK:=r2.going_to);
	r2.going_to_f_trig(CLK:=r2.going_to);
	r2.going_to_os := r2.going_to_r_trig.Q;
	r2.going_to_ns := r2.going_to_f_trig.Q;

	r3.fire_r_trig(CLK:=r3.fire);
	r3.fire_f_trig(CLK:=r3.fire);
	r3.fire_os := r3.fire_r_trig.Q;
	r3.fire_ns := r3.fire_f_trig.Q;
	r3.going_to_r_trig(CLK:=r3.going_to);
	r3.going_to_f_trig(CLK:=r3.going_to);
	r3.going_to_os := r3.going_to_r_trig.Q;
	r3.going_to_ns := r3.going_to_f_trig.Q;

	r4.fire_r_trig(CLK:=r4.fire);
	r4.fire_f_trig(CLK:=r4.fire);
	r4.fire_os := r4.fire_r_trig.Q;
	r4.fire_ns := r4.fire_f_trig.Q;
	r4.going_to_r_trig(CLK:=r4.going_to);
	r4.going_to_f_trig(CLK:=r4.going_to);
	r4.going_to_os := r4.going_to_r_trig.Q;
	r4.going_to_ns := r4.going_to_f_trig.Q;

	r5.fire_r_trig(CLK:=r5.fire);
	r5.fire_f_trig(CLK:=r5.fire);
	r5.fire_os := r5.fire_r_trig.Q;
	r5.fire_ns := r5.fire_f_trig.Q;
	r5.going_to_r_trig(CLK:=r5.going_to);
	r5.going_to_f_trig(CLK:=r5.going_to);
	r5.going_to_os := r5.going_to_r_trig.Q;
	r5.going_to_ns := r5.going_to_f_trig.Q;

	r6.fire_r_trig(CLK:=r6.fire);
	r6.fire_f_trig(CLK:=r6.fire);
	r6.fire_os := r6.fire_r_trig.Q;
	r6.fire_ns := r6.fire_f_trig.Q;
	r6.going_to_r_trig(CLK:=r6.going_to);
	r6.going_to_f_trig(CLK:=r6.going_to);
	r6.going_to_os := r6.going_to_r_trig.Q;
	r6.going_to_ns := r6.going_to_f_trig.Q;

	r7.fire_r_trig(CLK:=r7.fire);
	r7.fire_f_trig(CLK:=r7.fire);
	r7.fire_os := r7.fire_r_trig.Q;
	r7.fire_ns := r7.fire_f_trig.Q;
	r7.going_to_r_trig(CLK:=r7.going_to);
	r7.going_to_f_trig(CLK:=r7.going_to);
	r7.going_to_os := r7.going_to_r_trig.Q;
	r7.going_to_ns := r7.going_to_f_trig.Q;

	r8.fire_r_trig(CLK:=r8.fire);
	r8.fire_f_trig(CLK:=r8.fire);
	r8.fire_os := r8.fire_r_trig.Q;
	r8.fire_ns := r8.fire_f_trig.Q;
	r8.going_to_r_trig(CLK:=r8.going_to);
	r8.going_to_f_trig(CLK:=r8.going_to);
	r8.going_to_os := r8.going_to_r_trig.Q;
	r8.going_to_ns := r8.going_to_f_trig.Q;

	r9.fire_r_trig(CLK:=r9.fire);
	r9.fire_f_trig(CLK:=r9.fire);
	r9.fire_os := r9.fire_r_trig.Q;
	r9.fire_ns := r9.fire_f_trig.Q;
	r9.going_to_r_trig(CLK:=r9.going_to);
	r9.going_to_f_trig(CLK:=r9.going_to);
	r9.going_to_os := r9.going_to_r_trig.Q;
	r9.going_to_ns := r9.going_to_f_trig.Q;

	r10.fire_r_trig(CLK:=r10.fire);
	r10.fire_f_trig(CLK:=r10.fire);
	r10.fire_os := r10.fire_r_trig.Q;
	r10.fire_ns := r10.fire_f_trig.Q;
	r10.going_to_r_trig(CLK:=r10.going_to);
	r10.going_to_f_trig(CLK:=r10.going_to);
	r10.going_to_os := r10.going_to_r_trig.Q;
	r10.going_to_ns := r10.going_to_f_trig.Q;

	r11.fire_r_trig(CLK:=r11.fire);
	r11.fire_f_trig(CLK:=r11.fire);
	r11.fire_os := r11.fire_r_trig.Q;
	r11.fire_ns := r11.fire_f_trig.Q;
	r11.going_to_r_trig(CLK:=r11.going_to);
	r11.going_to_f_trig(CLK:=r11.going_to);
	r11.going_to_os := r11.going_to_r_trig.Q;
	r11.going_to_ns := r11.going_to_f_trig.Q;

	r12.fire_r_trig(CLK:=r12.fire);
	r12.fire_f_trig(CLK:=r12.fire);
	r12.fire_os := r12.fire_r_trig.Q;
	r12.fire_ns := r12.fire_f_trig.Q;
	r12.going_to_r_trig(CLK:=r12.going_to);
	r12.going_to_f_trig(CLK:=r12.going_to);
	r12.going_to_os := r12.going_to_r_trig.Q;
	r12.going_to_ns := r12.going_to_f_trig.Q;

	r13.fire_r_trig(CLK:=r13.fire);
	r13.fire_f_trig(CLK:=r13.fire);
	r13.fire_os := r13.fire_r_trig.Q;
	r13.fire_ns := r13.fire_f_trig.Q;
	r13.going_to_r_trig(CLK:=r13.going_to);
	r13.going_to_f_trig(CLK:=r13.going_to);
	r13.going_to_os := r13.going_to_r_trig.Q;
	r13.going_to_ns := r13.going_to_f_trig.Q;

	r14.fire_r_trig(CLK:=r14.fire);
	r14.fire_f_trig(CLK:=r14.fire);
	r14.fire_os := r14.fire_r_trig.Q;
	r14.fire_ns := r14.fire_f_trig.Q;
	r14.going_to_r_trig(CLK:=r14.going_to);
	r14.going_to_f_trig(CLK:=r14.going_to);
	r14.going_to_os := r14.going_to_r_trig.Q;
	r14.going_to_ns := r14.going_to_f_trig.Q;

	r15.fire_r_trig(CLK:=r15.fire);
	r15.fire_f_trig(CLK:=r15.fire);
	r15.fire_os := r15.fire_r_trig.Q;
	r15.fire_ns := r15.fire_f_trig.Q;
	r15.going_to_r_trig(CLK:=r15.going_to);
	r15.going_to_f_trig(CLK:=r15.going_to);
	r15.going_to_os := r15.going_to_r_trig.Q;
	r15.going_to_ns := r15.going_to_f_trig.Q;

	r16.fire_r_trig(CLK:=r16.fire);
	r16.fire_f_trig(CLK:=r16.fire);
	r16.fire_os := r16.fire_r_trig.Q;
	r16.fire_ns := r16.fire_f_trig.Q;
	r16.going_to_r_trig(CLK:=r16.going_to);
	r16.going_to_f_trig(CLK:=r16.going_to);
	r16.going_to_os := r16.going_to_r_trig.Q;
	r16.going_to_ns := r16.going_to_f_trig.Q;

	r17.fire_r_trig(CLK:=r17.fire);
	r17.fire_f_trig(CLK:=r17.fire);
	r17.fire_os := r17.fire_r_trig.Q;
	r17.fire_ns := r17.fire_f_trig.Q;
	r17.going_to_r_trig(CLK:=r17.going_to);
	r17.going_to_f_trig(CLK:=r17.going_to);
	r17.going_to_os := r17.going_to_r_trig.Q;
	r17.going_to_ns := r17.going_to_f_trig.Q;

	r18.fire_r_trig(CLK:=r18.fire);
	r18.fire_f_trig(CLK:=r18.fire);
	r18.fire_os := r18.fire_r_trig.Q;
	r18.fire_ns := r18.fire_f_trig.Q;
	r18.going_to_r_trig(CLK:=r18.going_to);
	r18.going_to_f_trig(CLK:=r18.going_to);
	r18.going_to_os := r18.going_to_r_trig.Q;
	r18.going_to_ns := r18.going_to_f_trig.Q;

	r19.fire_r_trig(CLK:=r19.fire);
	r19.fire_f_trig(CLK:=r19.fire);
	r19.fire_os := r19.fire_r_trig.Q;
	r19.fire_ns := r19.fire_f_trig.Q;
	r19.going_to_r_trig(CLK:=r19.going_to);
	r19.going_to_f_trig(CLK:=r19.going_to);
	r19.going_to_os := r19.going_to_r_trig.Q;
	r19.going_to_ns := r19.going_to_f_trig.Q;

	r20.fire_r_trig(CLK:=r20.fire);
	r20.fire_f_trig(CLK:=r20.fire);
	r20.fire_os := r20.fire_r_trig.Q;
	r20.fire_ns := r20.fire_f_trig.Q;
	r20.going_to_r_trig(CLK:=r20.going_to);
	r20.going_to_f_trig(CLK:=r20.going_to);
	r20.going_to_os := r20.going_to_r_trig.Q;
	r20.going_to_ns := r20.going_to_f_trig.Q;

	r21.fire_r_trig(CLK:=r21.fire);
	r21.fire_f_trig(CLK:=r21.fire);
	r21.fire_os := r21.fire_r_trig.Q;
	r21.fire_ns := r21.fire_f_trig.Q;
	r21.going_to_r_trig(CLK:=r21.going_to);
	r21.going_to_f_trig(CLK:=r21.going_to);
	r21.going_to_os := r21.going_to_r_trig.Q;
	r21.going_to_ns := r21.going_to_f_trig.Q;

	r22.fire_r_trig(CLK:=r22.fire);
	r22.fire_f_trig(CLK:=r22.fire);
	r22.fire_os := r22.fire_r_trig.Q;
	r22.fire_ns := r22.fire_f_trig.Q;
	r22.going_to_r_trig(CLK:=r22.going_to);
	r22.going_to_f_trig(CLK:=r22.going_to);
	r22.going_to_os := r22.going_to_r_trig.Q;
	r22.going_to_ns := r22.going_to_f_trig.Q;

	r23.fire_r_trig(CLK:=r23.fire);
	r23.fire_f_trig(CLK:=r23.fire);
	r23.fire_os := r23.fire_r_trig.Q;
	r23.fire_ns := r23.fire_f_trig.Q;
	r23.going_to_r_trig(CLK:=r23.going_to);
	r23.going_to_f_trig(CLK:=r23.going_to);
	r23.going_to_os := r23.going_to_r_trig.Q;
	r23.going_to_ns := r23.going_to_f_trig.Q;

	r24.fire_r_trig(CLK:=r24.fire);
	r24.fire_f_trig(CLK:=r24.fire);
	r24.fire_os := r24.fire_r_trig.Q;
	r24.fire_ns := r24.fire_f_trig.Q;
	r24.going_to_r_trig(CLK:=r24.going_to);
	r24.going_to_f_trig(CLK:=r24.going_to);
	r24.going_to_os := r24.going_to_r_trig.Q;
	r24.going_to_ns := r24.going_to_f_trig.Q;

	r25.fire_r_trig(CLK:=r25.fire);
	r25.fire_f_trig(CLK:=r25.fire);
	r25.fire_os := r25.fire_r_trig.Q;
	r25.fire_ns := r25.fire_f_trig.Q;
	r25.going_to_r_trig(CLK:=r25.going_to);
	r25.going_to_f_trig(CLK:=r25.going_to);
	r25.going_to_os := r25.going_to_r_trig.Q;
	r25.going_to_ns := r25.going_to_f_trig.Q;

	r26.fire_r_trig(CLK:=r26.fire);
	r26.fire_f_trig(CLK:=r26.fire);
	r26.fire_os := r26.fire_r_trig.Q;
	r26.fire_ns := r26.fire_f_trig.Q;
	r26.going_to_r_trig(CLK:=r26.going_to);
	r26.going_to_f_trig(CLK:=r26.going_to);
	r26.going_to_os := r26.going_to_r_trig.Q;
	r26.going_to_ns := r26.going_to_f_trig.Q;

	r27.fire_r_trig(CLK:=r27.fire);
	r27.fire_f_trig(CLK:=r27.fire);
	r27.fire_os := r27.fire_r_trig.Q;
	r27.fire_ns := r27.fire_f_trig.Q;
	r27.going_to_r_trig(CLK:=r27.going_to);
	r27.going_to_f_trig(CLK:=r27.going_to);
	r27.going_to_os := r27.going_to_r_trig.Q;
	r27.going_to_ns := r27.going_to_f_trig.Q;

	r28.fire_r_trig(CLK:=r28.fire);
	r28.fire_f_trig(CLK:=r28.fire);
	r28.fire_os := r28.fire_r_trig.Q;
	r28.fire_ns := r28.fire_f_trig.Q;
	r28.going_to_r_trig(CLK:=r28.going_to);
	r28.going_to_f_trig(CLK:=r28.going_to);
	r28.going_to_os := r28.going_to_r_trig.Q;
	r28.going_to_ns := r28.going_to_f_trig.Q;

	r29.fire_r_trig(CLK:=r29.fire);
	r29.fire_f_trig(CLK:=r29.fire);
	r29.fire_os := r29.fire_r_trig.Q;
	r29.fire_ns := r29.fire_f_trig.Q;
	r29.going_to_r_trig(CLK:=r29.going_to);
	r29.going_to_f_trig(CLK:=r29.going_to);
	r29.going_to_os := r29.going_to_r_trig.Q;
	r29.going_to_ns := r29.going_to_f_trig.Q;

	r30.fire_r_trig(CLK:=r30.fire);
	r30.fire_f_trig(CLK:=r30.fire);
	r30.fire_os := r30.fire_r_trig.Q;
	r30.fire_ns := r30.fire_f_trig.Q;
	r30.going_to_r_trig(CLK:=r30.going_to);
	r30.going_to_f_trig(CLK:=r30.going_to);
	r30.going_to_os := r30.going_to_r_trig.Q;
	r30.going_to_ns := r30.going_to_f_trig.Q;

	r31.fire_r_trig(CLK:=r31.fire);
	r31.fire_f_trig(CLK:=r31.fire);
	r31.fire_os := r31.fire_r_trig.Q;
	r31.fire_ns := r31.fire_f_trig.Q;
	r31.going_to_r_trig(CLK:=r31.going_to);
	r31.going_to_f_trig(CLK:=r31.going_to);
	r31.going_to_os := r31.going_to_r_trig.Q;
	r31.going_to_ns := r31.going_to_f_trig.Q;

	r32.fire_r_trig(CLK:=r32.fire);
	r32.fire_f_trig(CLK:=r32.fire);
	r32.fire_os := r32.fire_r_trig.Q;
	r32.fire_ns := r32.fire_f_trig.Q;
	r32.going_to_r_trig(CLK:=r32.going_to);
	r32.going_to_f_trig(CLK:=r32.going_to);
	r32.going_to_os := r32.going_to_r_trig.Q;
	r32.going_to_ns := r32.going_to_f_trig.Q;

	r33.fire_r_trig(CLK:=r33.fire);
	r33.fire_f_trig(CLK:=r33.fire);
	r33.fire_os := r33.fire_r_trig.Q;
	r33.fire_ns := r33.fire_f_trig.Q;
	r33.going_to_r_trig(CLK:=r33.going_to);
	r33.going_to_f_trig(CLK:=r33.going_to);
	r33.going_to_os := r33.going_to_r_trig.Q;
	r33.going_to_ns := r33.going_to_f_trig.Q;

	r34.fire_r_trig(CLK:=r34.fire);
	r34.fire_f_trig(CLK:=r34.fire);
	r34.fire_os := r34.fire_r_trig.Q;
	r34.fire_ns := r34.fire_f_trig.Q;
	r34.going_to_r_trig(CLK:=r34.going_to);
	r34.going_to_f_trig(CLK:=r34.going_to);
	r34.going_to_os := r34.going_to_r_trig.Q;
	r34.going_to_ns := r34.going_to_f_trig.Q;

	r35.fire_r_trig(CLK:=r35.fire);
	r35.fire_f_trig(CLK:=r35.fire);
	r35.fire_os := r35.fire_r_trig.Q;
	r35.fire_ns := r35.fire_f_trig.Q;
	r35.going_to_r_trig(CLK:=r35.going_to);
	r35.going_to_f_trig(CLK:=r35.going_to);
	r35.going_to_os := r35.going_to_r_trig.Q;
	r35.going_to_ns := r35.going_to_f_trig.Q;

	r36.fire_r_trig(CLK:=r36.fire);
	r36.fire_f_trig(CLK:=r36.fire);
	r36.fire_os := r36.fire_r_trig.Q;
	r36.fire_ns := r36.fire_f_trig.Q;
	r36.going_to_r_trig(CLK:=r36.going_to);
	r36.going_to_f_trig(CLK:=r36.going_to);
	r36.going_to_os := r36.going_to_r_trig.Q;
	r36.going_to_ns := r36.going_to_f_trig.Q;

	r37.fire_r_trig(CLK:=r37.fire);
	r37.fire_f_trig(CLK:=r37.fire);
	r37.fire_os := r37.fire_r_trig.Q;
	r37.fire_ns := r37.fire_f_trig.Q;
	r37.going_to_r_trig(CLK:=r37.going_to);
	r37.going_to_f_trig(CLK:=r37.going_to);
	r37.going_to_os := r37.going_to_r_trig.Q;
	r37.going_to_ns := r37.going_to_f_trig.Q;

	r38.fire_r_trig(CLK:=r38.fire);
	r38.fire_f_trig(CLK:=r38.fire);
	r38.fire_os := r38.fire_r_trig.Q;
	r38.fire_ns := r38.fire_f_trig.Q;
	r38.going_to_r_trig(CLK:=r38.going_to);
	r38.going_to_f_trig(CLK:=r38.going_to);
	r38.going_to_os := r38.going_to_r_trig.Q;
	r38.going_to_ns := r38.going_to_f_trig.Q;

	r39.fire_r_trig(CLK:=r39.fire);
	r39.fire_f_trig(CLK:=r39.fire);
	r39.fire_os := r39.fire_r_trig.Q;
	r39.fire_ns := r39.fire_f_trig.Q;
	r39.going_to_r_trig(CLK:=r39.going_to);
	r39.going_to_f_trig(CLK:=r39.going_to);
	r39.going_to_os := r39.going_to_r_trig.Q;
	r39.going_to_ns := r39.going_to_f_trig.Q;

	r40.fire_r_trig(CLK:=r40.fire);
	r40.fire_f_trig(CLK:=r40.fire);
	r40.fire_os := r40.fire_r_trig.Q;
	r40.fire_ns := r40.fire_f_trig.Q;
	r40.going_to_r_trig(CLK:=r40.going_to);
	r40.going_to_f_trig(CLK:=r40.going_to);
	r40.going_to_os := r40.going_to_r_trig.Q;
	r40.going_to_ns := r40.going_to_f_trig.Q;

	r41.fire_r_trig(CLK:=r41.fire);
	r41.fire_f_trig(CLK:=r41.fire);
	r41.fire_os := r41.fire_r_trig.Q;
	r41.fire_ns := r41.fire_f_trig.Q;
	r41.going_to_r_trig(CLK:=r41.going_to);
	r41.going_to_f_trig(CLK:=r41.going_to);
	r41.going_to_os := r41.going_to_r_trig.Q;
	r41.going_to_ns := r41.going_to_f_trig.Q;

	r42.fire_r_trig(CLK:=r42.fire);
	r42.fire_f_trig(CLK:=r42.fire);
	r42.fire_os := r42.fire_r_trig.Q;
	r42.fire_ns := r42.fire_f_trig.Q;
	r42.going_to_r_trig(CLK:=r42.going_to);
	r42.going_to_f_trig(CLK:=r42.going_to);
	r42.going_to_os := r42.going_to_r_trig.Q;
	r42.going_to_ns := r42.going_to_f_trig.Q;

	r43.fire_r_trig(CLK:=r43.fire);
	r43.fire_f_trig(CLK:=r43.fire);
	r43.fire_os := r43.fire_r_trig.Q;
	r43.fire_ns := r43.fire_f_trig.Q;
	r43.going_to_r_trig(CLK:=r43.going_to);
	r43.going_to_f_trig(CLK:=r43.going_to);
	r43.going_to_os := r43.going_to_r_trig.Q;
	r43.going_to_ns := r43.going_to_f_trig.Q;

	r44.fire_r_trig(CLK:=r44.fire);
	r44.fire_f_trig(CLK:=r44.fire);
	r44.fire_os := r44.fire_r_trig.Q;
	r44.fire_ns := r44.fire_f_trig.Q;
	r44.going_to_r_trig(CLK:=r44.going_to);
	r44.going_to_f_trig(CLK:=r44.going_to);
	r44.going_to_os := r44.going_to_r_trig.Q;
	r44.going_to_ns := r44.going_to_f_trig.Q;

	r45.fire_r_trig(CLK:=r45.fire);
	r45.fire_f_trig(CLK:=r45.fire);
	r45.fire_os := r45.fire_r_trig.Q;
	r45.fire_ns := r45.fire_f_trig.Q;
	r45.going_to_r_trig(CLK:=r45.going_to);
	r45.going_to_f_trig(CLK:=r45.going_to);
	r45.going_to_os := r45.going_to_r_trig.Q;
	r45.going_to_ns := r45.going_to_f_trig.Q;

	r46.fire_r_trig(CLK:=r46.fire);
	r46.fire_f_trig(CLK:=r46.fire);
	r46.fire_os := r46.fire_r_trig.Q;
	r46.fire_ns := r46.fire_f_trig.Q;
	r46.going_to_r_trig(CLK:=r46.going_to);
	r46.going_to_f_trig(CLK:=r46.going_to);
	r46.going_to_os := r46.going_to_r_trig.Q;
	r46.going_to_ns := r46.going_to_f_trig.Q;

	r47.fire_r_trig(CLK:=r47.fire);
	r47.fire_f_trig(CLK:=r47.fire);
	r47.fire_os := r47.fire_r_trig.Q;
	r47.fire_ns := r47.fire_f_trig.Q;
	r47.going_to_r_trig(CLK:=r47.going_to);
	r47.going_to_f_trig(CLK:=r47.going_to);
	r47.going_to_os := r47.going_to_r_trig.Q;
	r47.going_to_ns := r47.going_to_f_trig.Q;

	r48.fire_r_trig(CLK:=r48.fire);
	r48.fire_f_trig(CLK:=r48.fire);
	r48.fire_os := r48.fire_r_trig.Q;
	r48.fire_ns := r48.fire_f_trig.Q;
	r48.going_to_r_trig(CLK:=r48.going_to);
	r48.going_to_f_trig(CLK:=r48.going_to);
	r48.going_to_os := r48.going_to_r_trig.Q;
	r48.going_to_ns := r48.going_to_f_trig.Q;

	r49.fire_r_trig(CLK:=r49.fire);
	r49.fire_f_trig(CLK:=r49.fire);
	r49.fire_os := r49.fire_r_trig.Q;
	r49.fire_ns := r49.fire_f_trig.Q;
	r49.going_to_r_trig(CLK:=r49.going_to);
	r49.going_to_f_trig(CLK:=r49.going_to);
	r49.going_to_os := r49.going_to_r_trig.Q;
	r49.going_to_ns := r49.going_to_f_trig.Q;

	r50.fire_r_trig(CLK:=r50.fire);
	r50.fire_f_trig(CLK:=r50.fire);
	r50.fire_os := r50.fire_r_trig.Q;
	r50.fire_ns := r50.fire_f_trig.Q;
	r50.going_to_r_trig(CLK:=r50.going_to);
	r50.going_to_f_trig(CLK:=r50.going_to);
	r50.going_to_os := r50.going_to_r_trig.Q;
	r50.going_to_ns := r50.going_to_f_trig.Q;

	r51.fire_r_trig(CLK:=r51.fire);
	r51.fire_f_trig(CLK:=r51.fire);
	r51.fire_os := r51.fire_r_trig.Q;
	r51.fire_ns := r51.fire_f_trig.Q;
	r51.going_to_r_trig(CLK:=r51.going_to);
	r51.going_to_f_trig(CLK:=r51.going_to);
	r51.going_to_os := r51.going_to_r_trig.Q;
	r51.going_to_ns := r51.going_to_f_trig.Q;

	r52.fire_r_trig(CLK:=r52.fire);
	r52.fire_f_trig(CLK:=r52.fire);
	r52.fire_os := r52.fire_r_trig.Q;
	r52.fire_ns := r52.fire_f_trig.Q;
	r52.going_to_r_trig(CLK:=r52.going_to);
	r52.going_to_f_trig(CLK:=r52.going_to);
	r52.going_to_os := r52.going_to_r_trig.Q;
	r52.going_to_ns := r52.going_to_f_trig.Q;

	r53.fire_r_trig(CLK:=r53.fire);
	r53.fire_f_trig(CLK:=r53.fire);
	r53.fire_os := r53.fire_r_trig.Q;
	r53.fire_ns := r53.fire_f_trig.Q;
	r53.going_to_r_trig(CLK:=r53.going_to);
	r53.going_to_f_trig(CLK:=r53.going_to);
	r53.going_to_os := r53.going_to_r_trig.Q;
	r53.going_to_ns := r53.going_to_f_trig.Q;

	r54.fire_r_trig(CLK:=r54.fire);
	r54.fire_f_trig(CLK:=r54.fire);
	r54.fire_os := r54.fire_r_trig.Q;
	r54.fire_ns := r54.fire_f_trig.Q;
	r54.going_to_r_trig(CLK:=r54.going_to);
	r54.going_to_f_trig(CLK:=r54.going_to);
	r54.going_to_os := r54.going_to_r_trig.Q;
	r54.going_to_ns := r54.going_to_f_trig.Q;

	r55.fire_r_trig(CLK:=r55.fire);
	r55.fire_f_trig(CLK:=r55.fire);
	r55.fire_os := r55.fire_r_trig.Q;
	r55.fire_ns := r55.fire_f_trig.Q;
	r55.going_to_r_trig(CLK:=r55.going_to);
	r55.going_to_f_trig(CLK:=r55.going_to);
	r55.going_to_os := r55.going_to_r_trig.Q;
	r55.going_to_ns := r55.going_to_f_trig.Q;

	r56.fire_r_trig(CLK:=r56.fire);
	r56.fire_f_trig(CLK:=r56.fire);
	r56.fire_os := r56.fire_r_trig.Q;
	r56.fire_ns := r56.fire_f_trig.Q;
	r56.going_to_r_trig(CLK:=r56.going_to);
	r56.going_to_f_trig(CLK:=r56.going_to);
	r56.going_to_os := r56.going_to_r_trig.Q;
	r56.going_to_ns := r56.going_to_f_trig.Q;

	r57.fire_r_trig(CLK:=r57.fire);
	r57.fire_f_trig(CLK:=r57.fire);
	r57.fire_os := r57.fire_r_trig.Q;
	r57.fire_ns := r57.fire_f_trig.Q;
	r57.going_to_r_trig(CLK:=r57.going_to);
	r57.going_to_f_trig(CLK:=r57.going_to);
	r57.going_to_os := r57.going_to_r_trig.Q;
	r57.going_to_ns := r57.going_to_f_trig.Q;

	r58.fire_r_trig(CLK:=r58.fire);
	r58.fire_f_trig(CLK:=r58.fire);
	r58.fire_os := r58.fire_r_trig.Q;
	r58.fire_ns := r58.fire_f_trig.Q;
	r58.going_to_r_trig(CLK:=r58.going_to);
	r58.going_to_f_trig(CLK:=r58.going_to);
	r58.going_to_os := r58.going_to_r_trig.Q;
	r58.going_to_ns := r58.going_to_f_trig.Q;

	r59.fire_r_trig(CLK:=r59.fire);
	r59.fire_f_trig(CLK:=r59.fire);
	r59.fire_os := r59.fire_r_trig.Q;
	r59.fire_ns := r59.fire_f_trig.Q;
	r59.going_to_r_trig(CLK:=r59.going_to);
	r59.going_to_f_trig(CLK:=r59.going_to);
	r59.going_to_os := r59.going_to_r_trig.Q;
	r59.going_to_ns := r59.going_to_f_trig.Q;

	r60.fire_r_trig(CLK:=r60.fire);
	r60.fire_f_trig(CLK:=r60.fire);
	r60.fire_os := r60.fire_r_trig.Q;
	r60.fire_ns := r60.fire_f_trig.Q;
	r60.going_to_r_trig(CLK:=r60.going_to);
	r60.going_to_f_trig(CLK:=r60.going_to);
	r60.going_to_os := r60.going_to_r_trig.Q;
	r60.going_to_ns := r60.going_to_f_trig.Q;

	r61.fire_r_trig(CLK:=r61.fire);
	r61.fire_f_trig(CLK:=r61.fire);
	r61.fire_os := r61.fire_r_trig.Q;
	r61.fire_ns := r61.fire_f_trig.Q;
	r61.going_to_r_trig(CLK:=r61.going_to);
	r61.going_to_f_trig(CLK:=r61.going_to);
	r61.going_to_os := r61.going_to_r_trig.Q;
	r61.going_to_ns := r61.going_to_f_trig.Q;

	r62.fire_r_trig(CLK:=r62.fire);
	r62.fire_f_trig(CLK:=r62.fire);
	r62.fire_os := r62.fire_r_trig.Q;
	r62.fire_ns := r62.fire_f_trig.Q;
	r62.going_to_r_trig(CLK:=r62.going_to);
	r62.going_to_f_trig(CLK:=r62.going_to);
	r62.going_to_os := r62.going_to_r_trig.Q;
	r62.going_to_ns := r62.going_to_f_trig.Q;

	r63.fire_r_trig(CLK:=r63.fire);
	r63.fire_f_trig(CLK:=r63.fire);
	r63.fire_os := r63.fire_r_trig.Q;
	r63.fire_ns := r63.fire_f_trig.Q;
	r63.going_to_r_trig(CLK:=r63.going_to);
	r63.going_to_f_trig(CLK:=r63.going_to);
	r63.going_to_os := r63.going_to_r_trig.Q;
	r63.going_to_ns := r63.going_to_f_trig.Q;

	r64.fire_r_trig(CLK:=r64.fire);
	r64.fire_f_trig(CLK:=r64.fire);
	r64.fire_os := r64.fire_r_trig.Q;
	r64.fire_ns := r64.fire_f_trig.Q;
	r64.going_to_r_trig(CLK:=r64.going_to);
	r64.going_to_f_trig(CLK:=r64.going_to);
	r64.going_to_os := r64.going_to_r_trig.Q;
	r64.going_to_ns := r64.going_to_f_trig.Q;

	r65.fire_r_trig(CLK:=r65.fire);
	r65.fire_f_trig(CLK:=r65.fire);
	r65.fire_os := r65.fire_r_trig.Q;
	r65.fire_ns := r65.fire_f_trig.Q;
	r65.going_to_r_trig(CLK:=r65.going_to);
	r65.going_to_f_trig(CLK:=r65.going_to);
	r65.going_to_os := r65.going_to_r_trig.Q;
	r65.going_to_ns := r65.going_to_f_trig.Q;

	r66.fire_r_trig(CLK:=r66.fire);
	r66.fire_f_trig(CLK:=r66.fire);
	r66.fire_os := r66.fire_r_trig.Q;
	r66.fire_ns := r66.fire_f_trig.Q;
	r66.going_to_r_trig(CLK:=r66.going_to);
	r66.going_to_f_trig(CLK:=r66.going_to);
	r66.going_to_os := r66.going_to_r_trig.Q;
	r66.going_to_ns := r66.going_to_f_trig.Q;

	r67.fire_r_trig(CLK:=r67.fire);
	r67.fire_f_trig(CLK:=r67.fire);
	r67.fire_os := r67.fire_r_trig.Q;
	r67.fire_ns := r67.fire_f_trig.Q;
	r67.going_to_r_trig(CLK:=r67.going_to);
	r67.going_to_f_trig(CLK:=r67.going_to);
	r67.going_to_os := r67.going_to_r_trig.Q;
	r67.going_to_ns := r67.going_to_f_trig.Q;

	r68.fire_r_trig(CLK:=r68.fire);
	r68.fire_f_trig(CLK:=r68.fire);
	r68.fire_os := r68.fire_r_trig.Q;
	r68.fire_ns := r68.fire_f_trig.Q;
	r68.going_to_r_trig(CLK:=r68.going_to);
	r68.going_to_f_trig(CLK:=r68.going_to);
	r68.going_to_os := r68.going_to_r_trig.Q;
	r68.going_to_ns := r68.going_to_f_trig.Q;

	r69.fire_r_trig(CLK:=r69.fire);
	r69.fire_f_trig(CLK:=r69.fire);
	r69.fire_os := r69.fire_r_trig.Q;
	r69.fire_ns := r69.fire_f_trig.Q;
	r69.going_to_r_trig(CLK:=r69.going_to);
	r69.going_to_f_trig(CLK:=r69.going_to);
	r69.going_to_os := r69.going_to_r_trig.Q;
	r69.going_to_ns := r69.going_to_f_trig.Q;

	r70.fire_r_trig(CLK:=r70.fire);
	r70.fire_f_trig(CLK:=r70.fire);
	r70.fire_os := r70.fire_r_trig.Q;
	r70.fire_ns := r70.fire_f_trig.Q;
	r70.going_to_r_trig(CLK:=r70.going_to);
	r70.going_to_f_trig(CLK:=r70.going_to);
	r70.going_to_os := r70.going_to_r_trig.Q;
	r70.going_to_ns := r70.going_to_f_trig.Q;

	r71.fire_r_trig(CLK:=r71.fire);
	r71.fire_f_trig(CLK:=r71.fire);
	r71.fire_os := r71.fire_r_trig.Q;
	r71.fire_ns := r71.fire_f_trig.Q;
	r71.going_to_r_trig(CLK:=r71.going_to);
	r71.going_to_f_trig(CLK:=r71.going_to);
	r71.going_to_os := r71.going_to_r_trig.Q;
	r71.going_to_ns := r71.going_to_f_trig.Q;

	r72.fire_r_trig(CLK:=r72.fire);
	r72.fire_f_trig(CLK:=r72.fire);
	r72.fire_os := r72.fire_r_trig.Q;
	r72.fire_ns := r72.fire_f_trig.Q;
	r72.going_to_r_trig(CLK:=r72.going_to);
	r72.going_to_f_trig(CLK:=r72.going_to);
	r72.going_to_os := r72.going_to_r_trig.Q;
	r72.going_to_ns := r72.going_to_f_trig.Q;

	r73.fire_r_trig(CLK:=r73.fire);
	r73.fire_f_trig(CLK:=r73.fire);
	r73.fire_os := r73.fire_r_trig.Q;
	r73.fire_ns := r73.fire_f_trig.Q;
	r73.going_to_r_trig(CLK:=r73.going_to);
	r73.going_to_f_trig(CLK:=r73.going_to);
	r73.going_to_os := r73.going_to_r_trig.Q;
	r73.going_to_ns := r73.going_to_f_trig.Q;

	r74.fire_r_trig(CLK:=r74.fire);
	r74.fire_f_trig(CLK:=r74.fire);
	r74.fire_os := r74.fire_r_trig.Q;
	r74.fire_ns := r74.fire_f_trig.Q;
	r74.going_to_r_trig(CLK:=r74.going_to);
	r74.going_to_f_trig(CLK:=r74.going_to);
	r74.going_to_os := r74.going_to_r_trig.Q;
	r74.going_to_ns := r74.going_to_f_trig.Q;

END_PROGRAM
```

#### RAIL_SUB.ld - not listed in the package file held
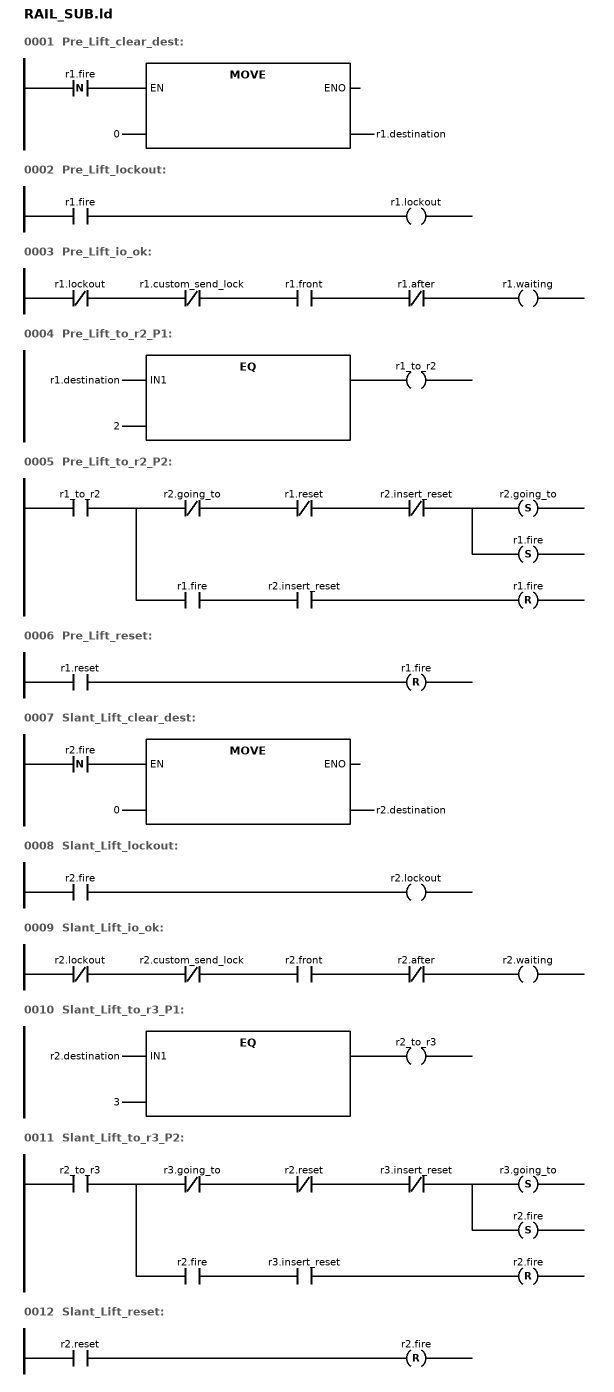
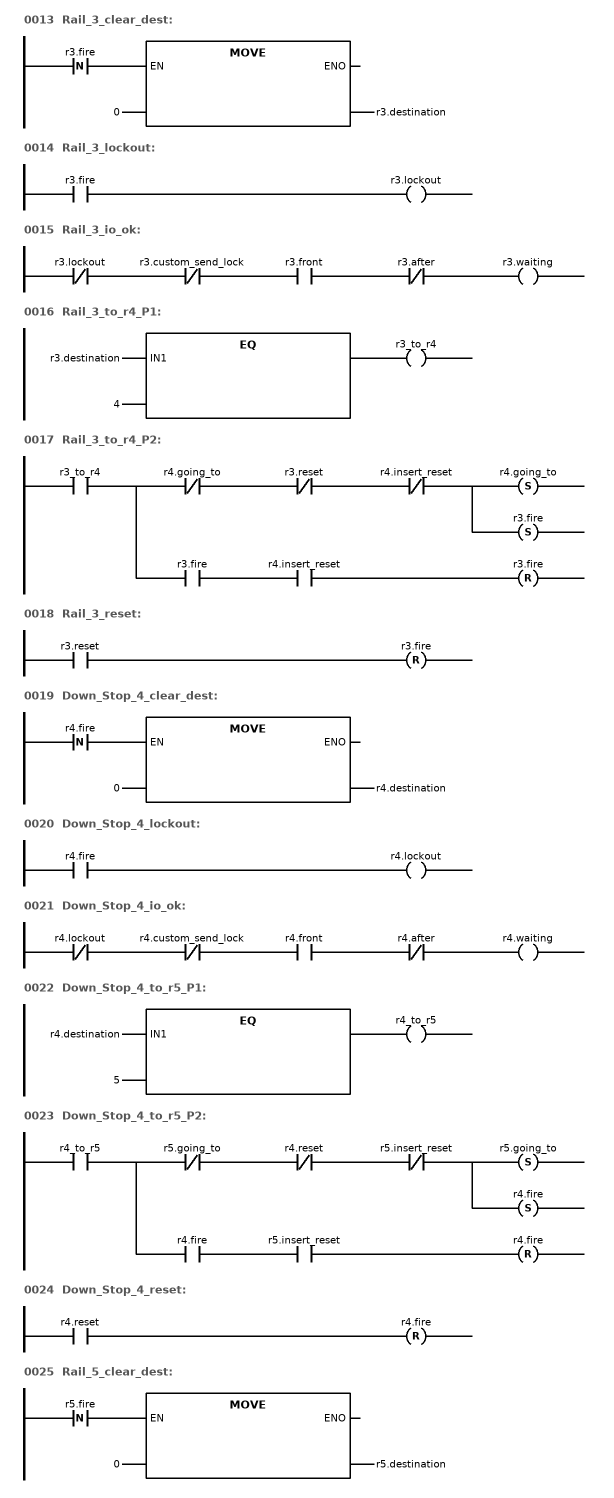
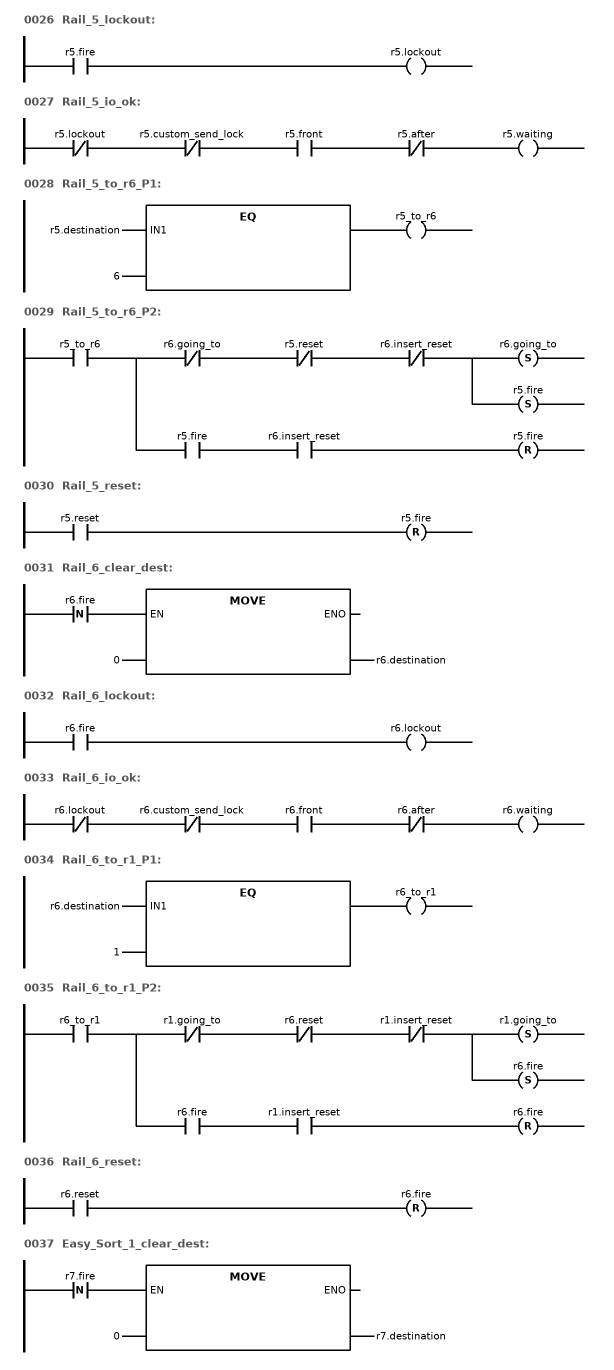
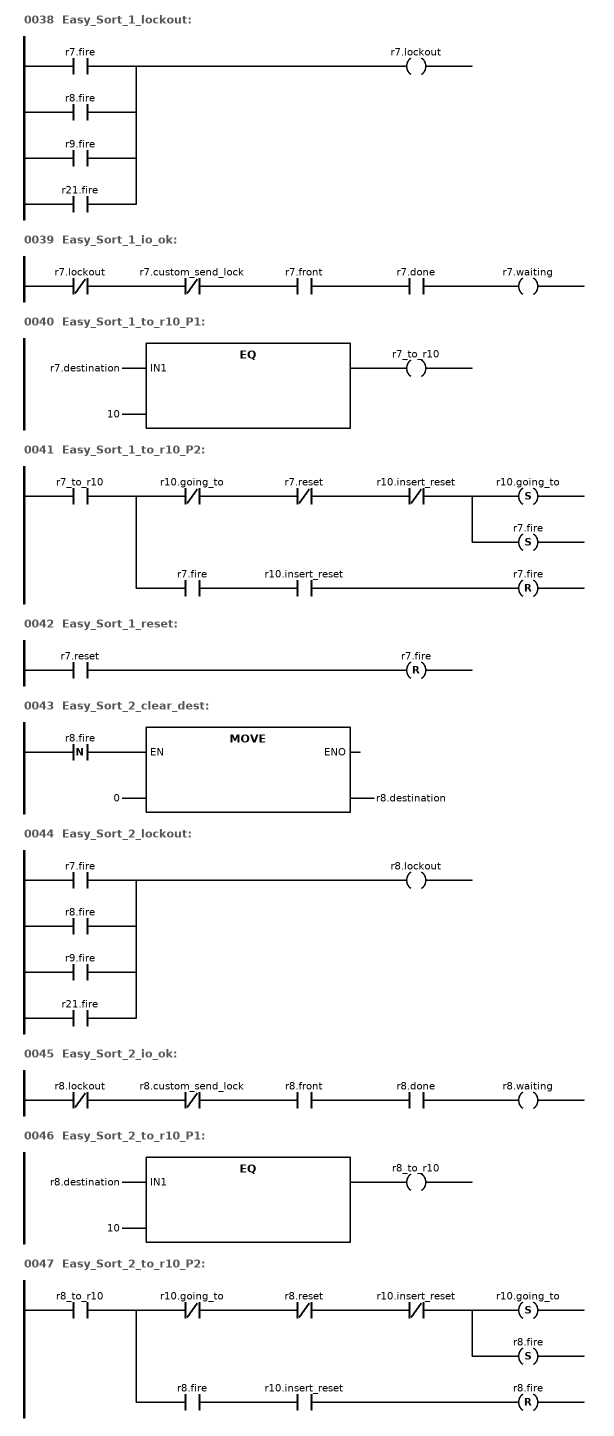
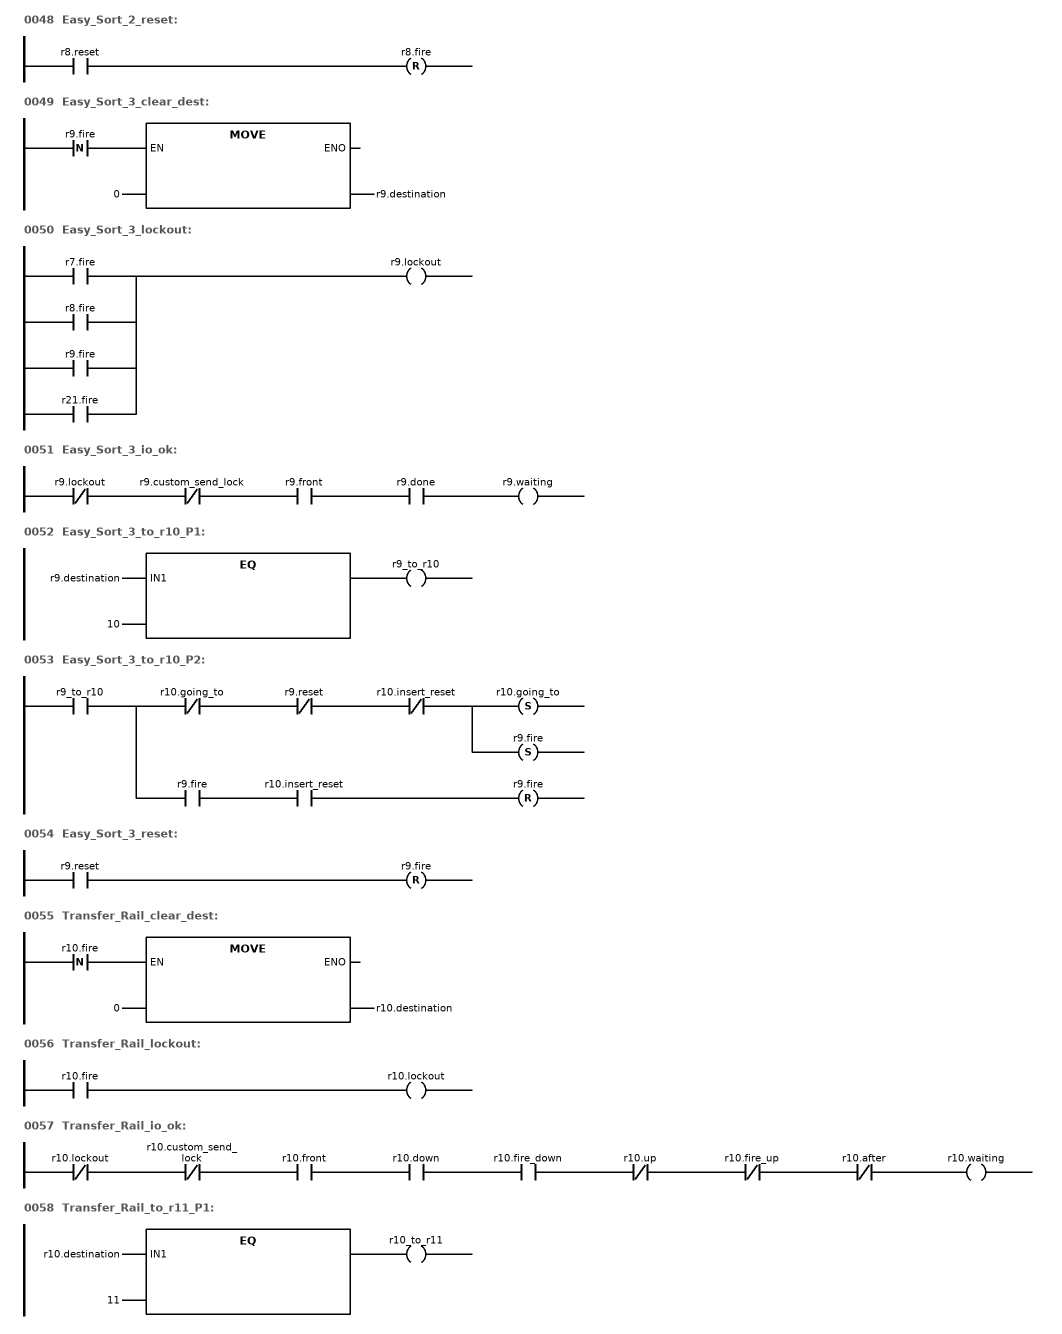
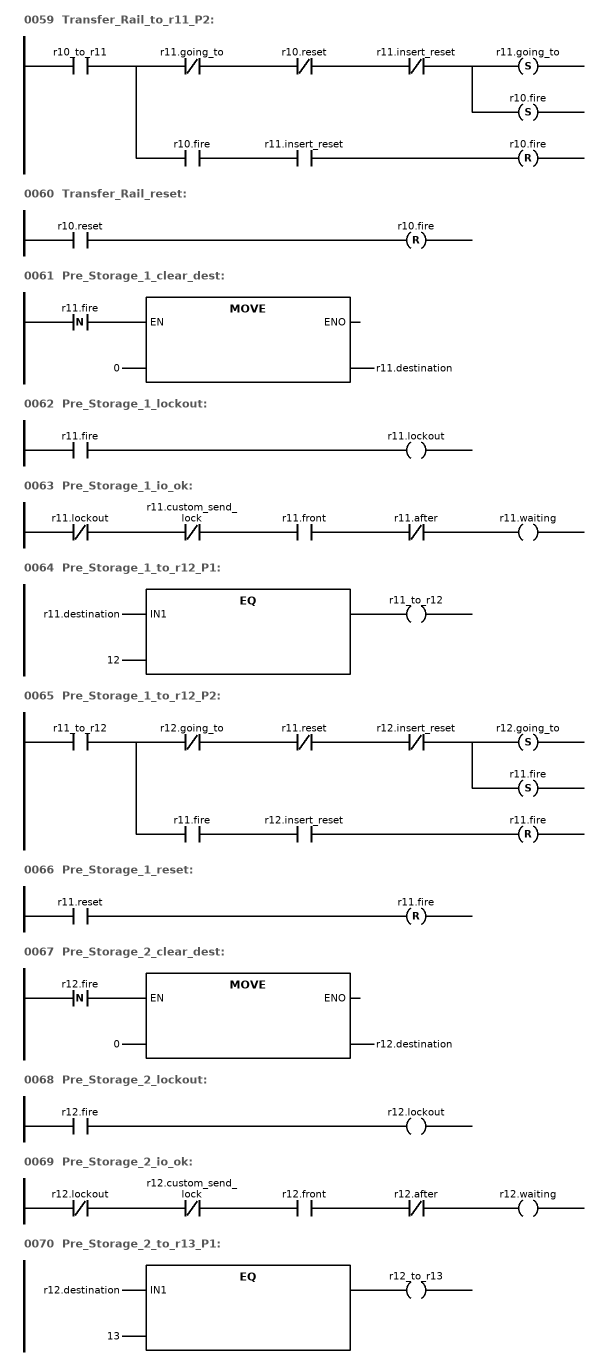
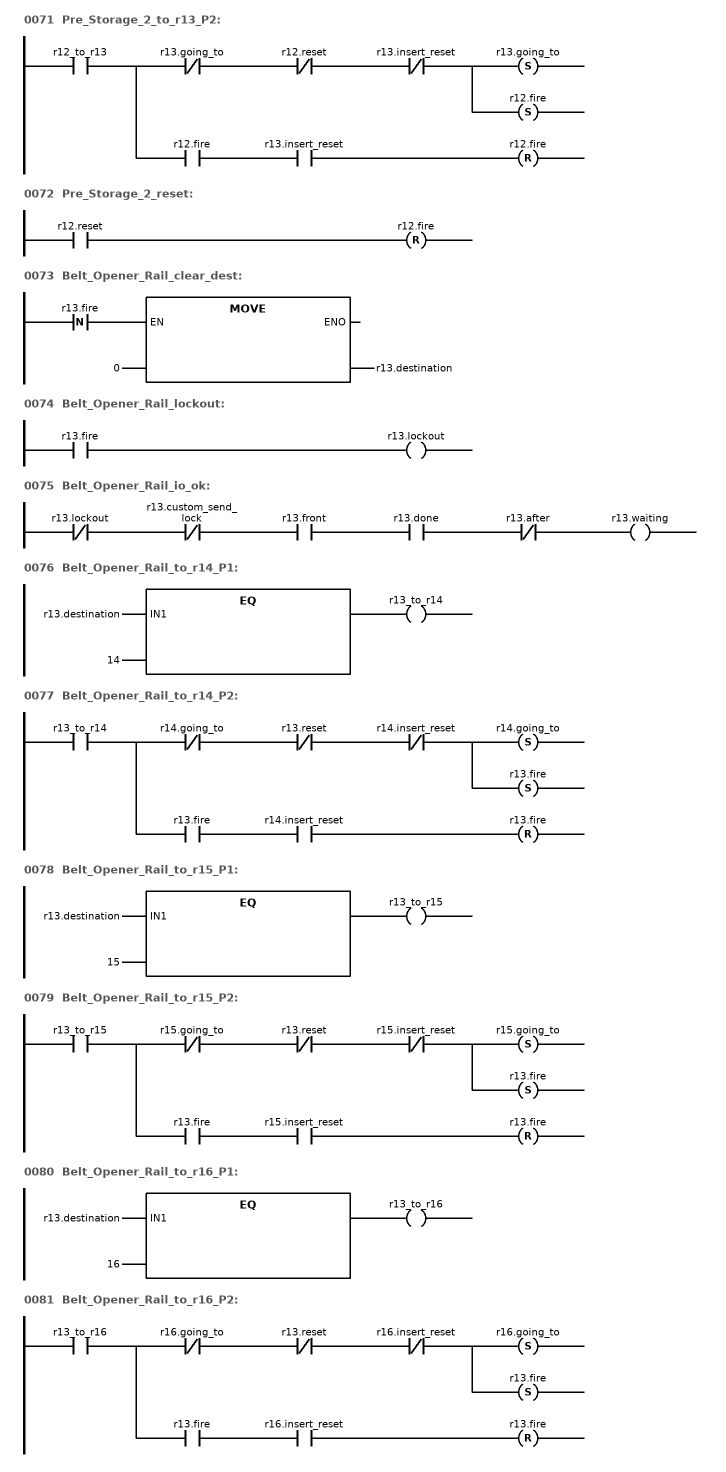
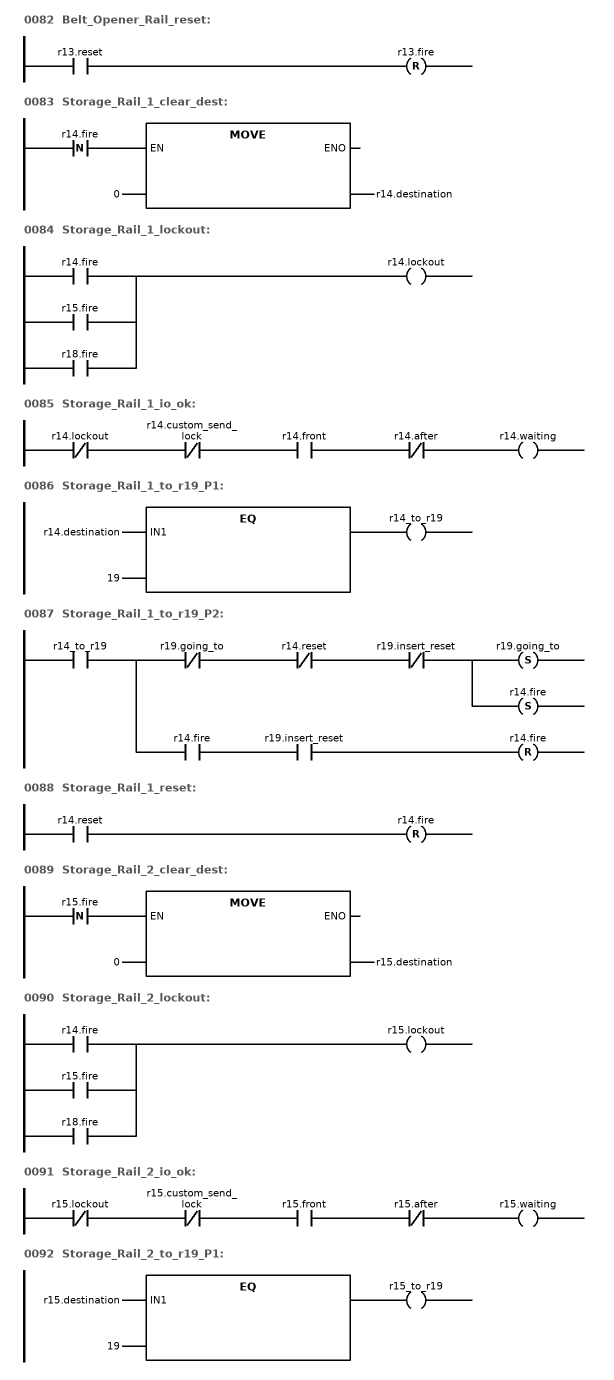
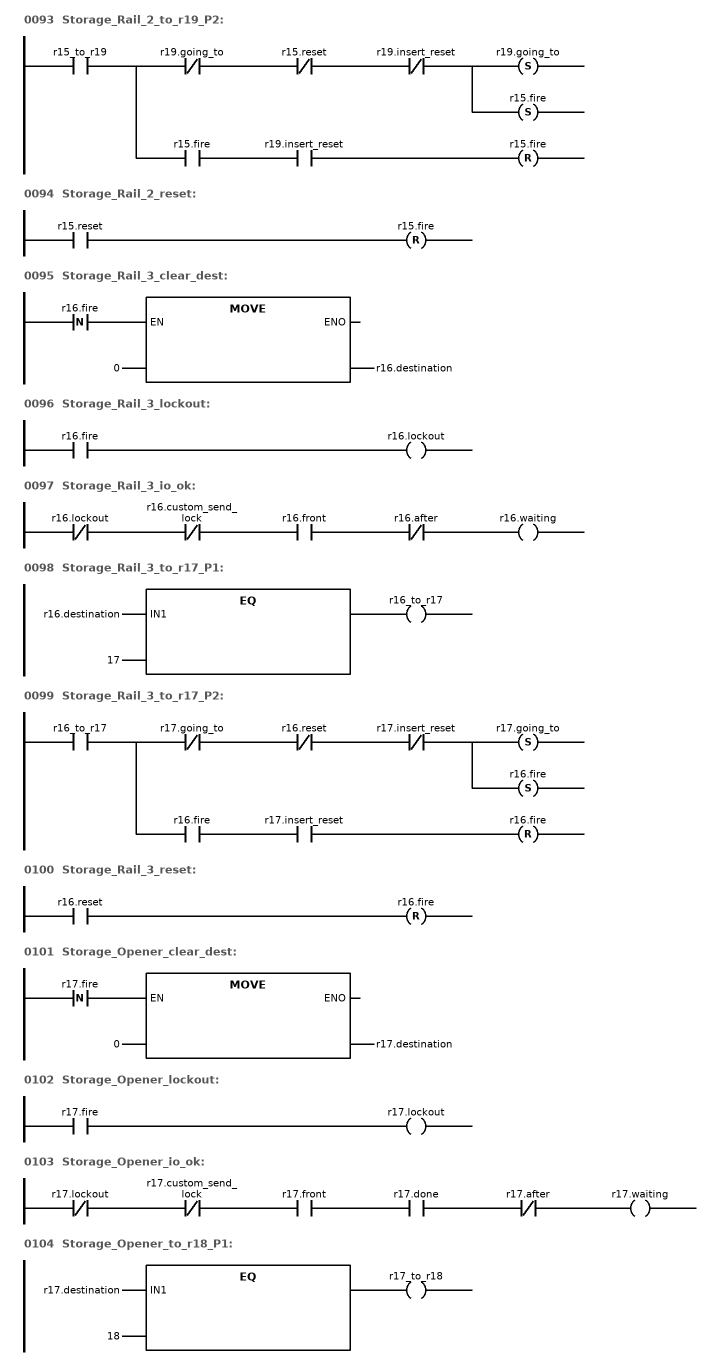
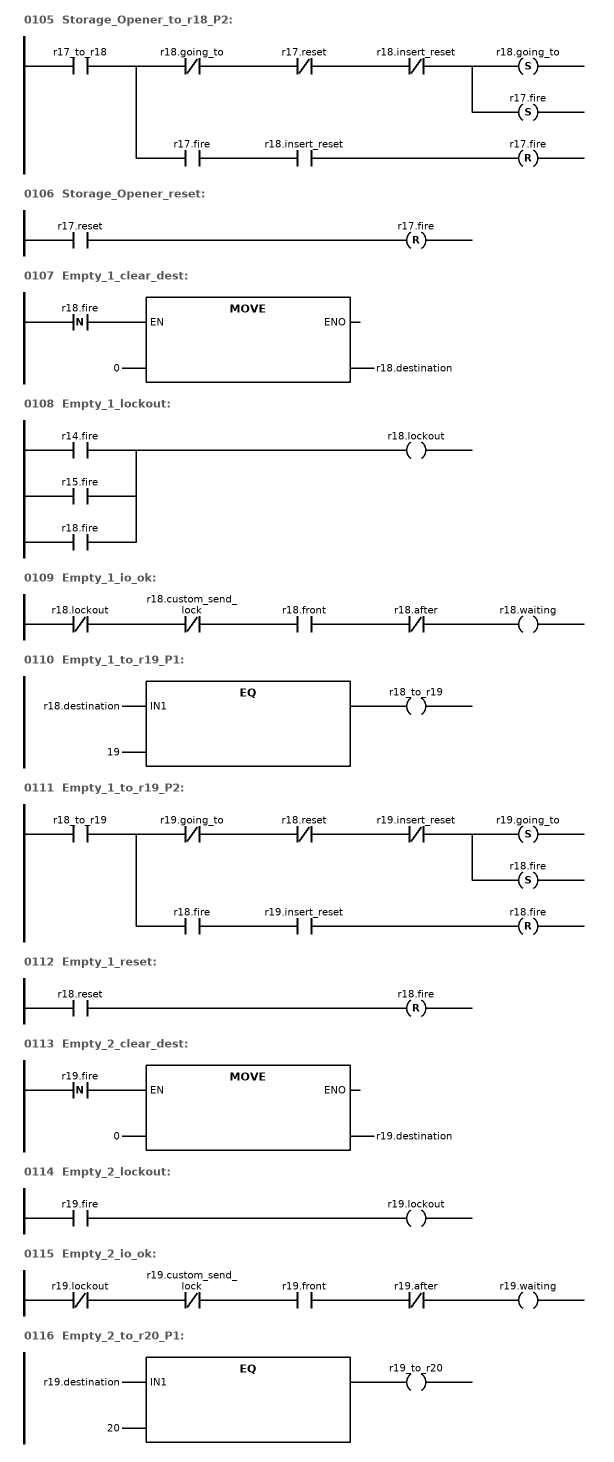
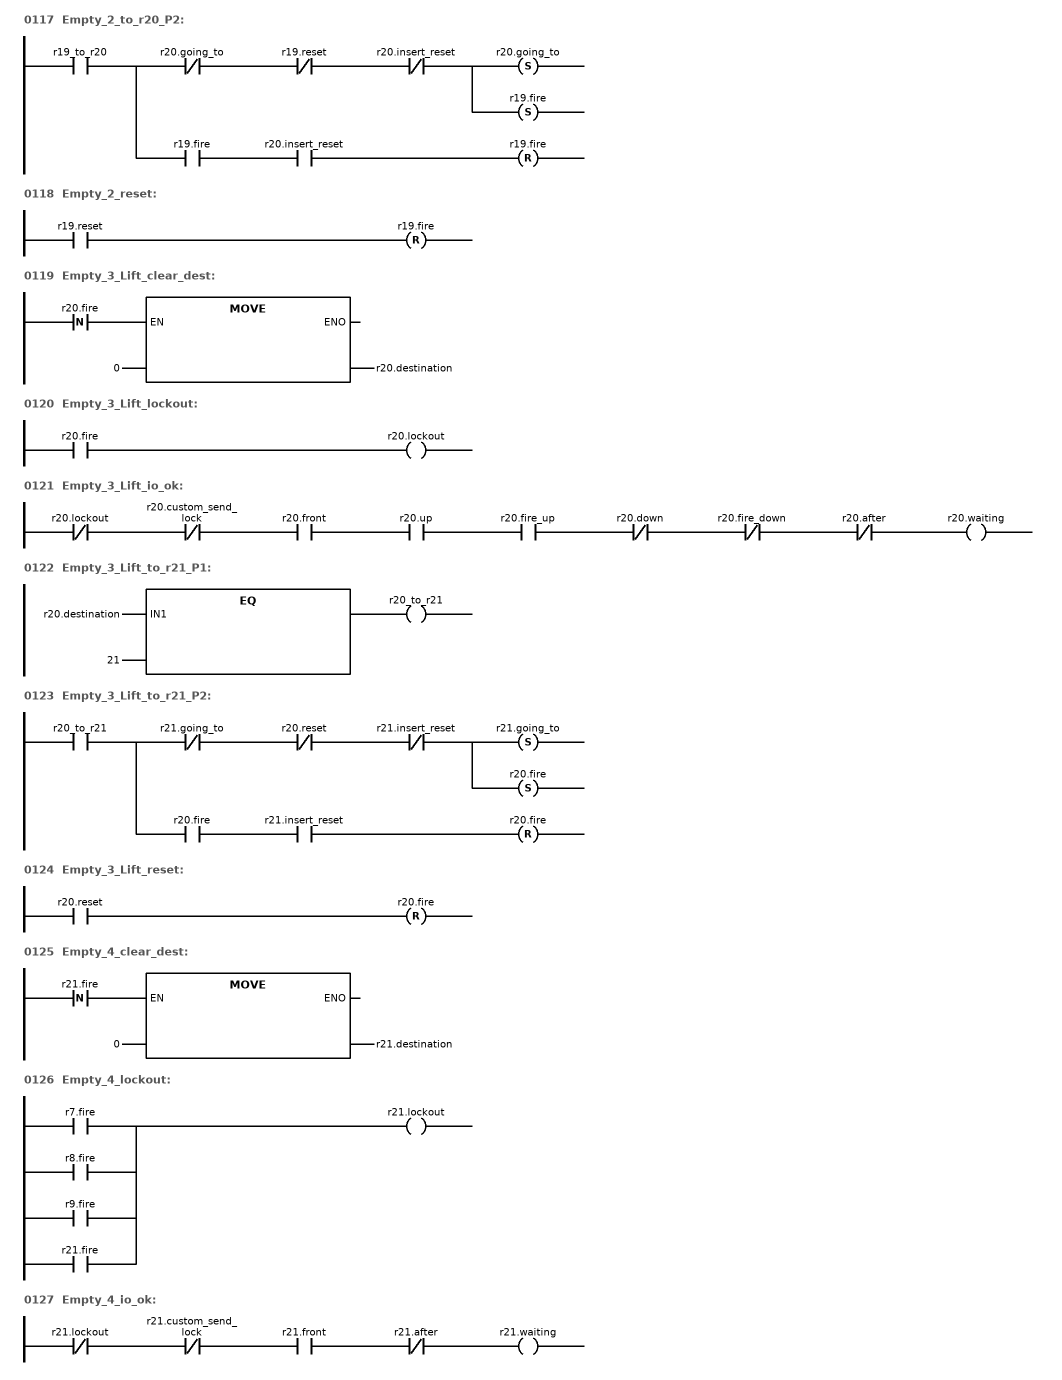
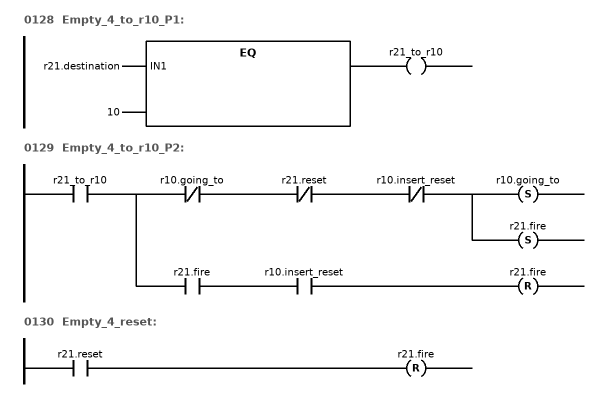
Ladder, written as Structured Text:
```iecst
PROGRAM _CYCLIC
VAR
    _e1 : F_TRIG;
    _p2 : BOOL;
    _e3 : F_TRIG;
    _p4 : BOOL;
    _e5 : F_TRIG;
    _p6 : BOOL;
    _e7 : F_TRIG;
    _p8 : BOOL;
    _e9 : F_TRIG;
    _p10 : BOOL;
    _e11 : F_TRIG;
    _p12 : BOOL;
    _e13 : F_TRIG;
    _p14 : BOOL;
    _e15 : F_TRIG;
    _p16 : BOOL;
    _e17 : F_TRIG;
    _p18 : BOOL;
    _e19 : F_TRIG;
    _p20 : BOOL;
    _e21 : F_TRIG;
    _p22 : BOOL;
    _e23 : F_TRIG;
    _p24 : BOOL;
    _e25 : F_TRIG;
    _p26 : BOOL;
    _p27 : BOOL;
    _p28 : BOOL;
    _e29 : F_TRIG;
    _p30 : BOOL;
    _e31 : F_TRIG;
    _p32 : BOOL;
    _e33 : F_TRIG;
    _p34 : BOOL;
    _e35 : F_TRIG;
    _p36 : BOOL;
    _e37 : F_TRIG;
    _p38 : BOOL;
    _e39 : F_TRIG;
    _p40 : BOOL;
    _e41 : F_TRIG;
    _p42 : BOOL;
    _e43 : F_TRIG;
    _p44 : BOOL;
END_VAR
(* Network 1 *)
Pre_Lift_clear_dest:
_e1(CLK := r1.fire);
IF _e1.Q THEN r1.destination := 0; END_IF;

(* Network 2 *)
Pre_Lift_lockout:
r1.lockout := r1.fire;

(* Network 3 *)
Pre_Lift_io_ok:
r1.waiting := NOT r1.lockout AND NOT r1.custom_send_lock AND r1.front AND NOT r1.after;

(* Network 4 *)
Pre_Lift_to_r2_P1:
r1_to_r2 := r1.destination = 2;

(* Network 5 *)
Pre_Lift_to_r2_P2:
_p2 := r1_to_r2 AND NOT r2.going_to AND NOT r1.reset AND NOT r2.insert_reset;
IF _p2 THEN
    r2.going_to := TRUE;
    r1.fire := TRUE;
END_IF;
IF r1_to_r2 AND r1.fire AND r2.insert_reset THEN r1.fire := FALSE; END_IF;

(* Network 6 *)
Pre_Lift_reset:
IF r1.reset THEN r1.fire := FALSE; END_IF;

(* Network 7 *)
Slant_Lift_clear_dest:
_e3(CLK := r2.fire);
IF _e3.Q THEN r2.destination := 0; END_IF;

(* Network 8 *)
Slant_Lift_lockout:
r2.lockout := r2.fire;

(* Network 9 *)
Slant_Lift_io_ok:
r2.waiting := NOT r2.lockout AND NOT r2.custom_send_lock AND r2.front AND NOT r2.after;

(* Network 10 *)
Slant_Lift_to_r3_P1:
r2_to_r3 := r2.destination = 3;

(* Network 11 *)
Slant_Lift_to_r3_P2:
_p4 := r2_to_r3 AND NOT r3.going_to AND NOT r2.reset AND NOT r3.insert_reset;
IF _p4 THEN
    r3.going_to := TRUE;
    r2.fire := TRUE;
END_IF;
IF r2_to_r3 AND r2.fire AND r3.insert_reset THEN r2.fire := FALSE; END_IF;

(* Network 12 *)
Slant_Lift_reset:
IF r2.reset THEN r2.fire := FALSE; END_IF;

(* Network 13 *)
Rail_3_clear_dest:
_e5(CLK := r3.fire);
IF _e5.Q THEN r3.destination := 0; END_IF;

(* Network 14 *)
Rail_3_lockout:
r3.lockout := r3.fire;

(* Network 15 *)
Rail_3_io_ok:
r3.waiting := NOT r3.lockout AND NOT r3.custom_send_lock AND r3.front AND NOT r3.after;

(* Network 16 *)
Rail_3_to_r4_P1:
r3_to_r4 := r3.destination = 4;

(* Network 17 *)
Rail_3_to_r4_P2:
_p6 := r3_to_r4 AND NOT r4.going_to AND NOT r3.reset AND NOT r4.insert_reset;
IF _p6 THEN
    r4.going_to := TRUE;
    r3.fire := TRUE;
END_IF;
IF r3_to_r4 AND r3.fire AND r4.insert_reset THEN r3.fire := FALSE; END_IF;

(* Network 18 *)
Rail_3_reset:
IF r3.reset THEN r3.fire := FALSE; END_IF;

(* Network 19 *)
Down_Stop_4_clear_dest:
_e7(CLK := r4.fire);
IF _e7.Q THEN r4.destination := 0; END_IF;

(* Network 20 *)
Down_Stop_4_lockout:
r4.lockout := r4.fire;

(* Network 21 *)
Down_Stop_4_io_ok:
r4.waiting := NOT r4.lockout AND NOT r4.custom_send_lock AND r4.front AND NOT r4.after;

(* Network 22 *)
Down_Stop_4_to_r5_P1:
r4_to_r5 := r4.destination = 5;

(* Network 23 *)
Down_Stop_4_to_r5_P2:
_p8 := r4_to_r5 AND NOT r5.going_to AND NOT r4.reset AND NOT r5.insert_reset;
IF _p8 THEN
    r5.going_to := TRUE;
    r4.fire := TRUE;
END_IF;
IF r4_to_r5 AND r4.fire AND r5.insert_reset THEN r4.fire := FALSE; END_IF;

(* Network 24 *)
Down_Stop_4_reset:
IF r4.reset THEN r4.fire := FALSE; END_IF;

(* Network 25 *)
Rail_5_clear_dest:
_e9(CLK := r5.fire);
IF _e9.Q THEN r5.destination := 0; END_IF;

(* Network 26 *)
Rail_5_lockout:
r5.lockout := r5.fire;

(* Network 27 *)
Rail_5_io_ok:
r5.waiting := NOT r5.lockout AND NOT r5.custom_send_lock AND r5.front AND NOT r5.after;

(* Network 28 *)
Rail_5_to_r6_P1:
r5_to_r6 := r5.destination = 6;

(* Network 29 *)
Rail_5_to_r6_P2:
_p10 := r5_to_r6 AND NOT r6.going_to AND NOT r5.reset AND NOT r6.insert_reset;
IF _p10 THEN
    r6.going_to := TRUE;
    r5.fire := TRUE;
END_IF;
IF r5_to_r6 AND r5.fire AND r6.insert_reset THEN r5.fire := FALSE; END_IF;

(* Network 30 *)
Rail_5_reset:
IF r5.reset THEN r5.fire := FALSE; END_IF;

(* Network 31 *)
Rail_6_clear_dest:
_e11(CLK := r6.fire);
IF _e11.Q THEN r6.destination := 0; END_IF;

(* Network 32 *)
Rail_6_lockout:
r6.lockout := r6.fire;

(* Network 33 *)
Rail_6_io_ok:
r6.waiting := NOT r6.lockout AND NOT r6.custom_send_lock AND r6.front AND NOT r6.after;

(* Network 34 *)
Rail_6_to_r1_P1:
r6_to_r1 := r6.destination = 1;

(* Network 35 *)
Rail_6_to_r1_P2:
_p12 := r6_to_r1 AND NOT r1.going_to AND NOT r6.reset AND NOT r1.insert_reset;
IF _p12 THEN
    r1.going_to := TRUE;
    r6.fire := TRUE;
END_IF;
IF r6_to_r1 AND r6.fire AND r1.insert_reset THEN r6.fire := FALSE; END_IF;

(* Network 36 *)
Rail_6_reset:
IF r6.reset THEN r6.fire := FALSE; END_IF;

(* Network 37 *)
Easy_Sort_1_clear_dest:
_e13(CLK := r7.fire);
IF _e13.Q THEN r7.destination := 0; END_IF;

(* Network 38 *)
Easy_Sort_1_lockout:
r7.lockout := r7.fire OR r8.fire OR r9.fire OR r21.fire;

(* Network 39 *)
Easy_Sort_1_io_ok:
r7.waiting := NOT r7.lockout AND NOT r7.custom_send_lock AND r7.front AND r7.done;

(* Network 40 *)
Easy_Sort_1_to_r10_P1:
r7_to_r10 := r7.destination = 10;

(* Network 41 *)
Easy_Sort_1_to_r10_P2:
_p14 := r7_to_r10 AND NOT r10.going_to AND NOT r7.reset AND NOT r10.insert_reset;
IF _p14 THEN
    r10.going_to := TRUE;
    r7.fire := TRUE;
END_IF;
IF r7_to_r10 AND r7.fire AND r10.insert_reset THEN r7.fire := FALSE; END_IF;

(* Network 42 *)
Easy_Sort_1_reset:
IF r7.reset THEN r7.fire := FALSE; END_IF;

(* Network 43 *)
Easy_Sort_2_clear_dest:
_e15(CLK := r8.fire);
IF _e15.Q THEN r8.destination := 0; END_IF;

(* Network 44 *)
Easy_Sort_2_lockout:
r8.lockout := r7.fire OR r8.fire OR r9.fire OR r21.fire;

(* Network 45 *)
Easy_Sort_2_io_ok:
r8.waiting := NOT r8.lockout AND NOT r8.custom_send_lock AND r8.front AND r8.done;

(* Network 46 *)
Easy_Sort_2_to_r10_P1:
r8_to_r10 := r8.destination = 10;

(* Network 47 *)
Easy_Sort_2_to_r10_P2:
_p16 := r8_to_r10 AND NOT r10.going_to AND NOT r8.reset AND NOT r10.insert_reset;
IF _p16 THEN
    r10.going_to := TRUE;
    r8.fire := TRUE;
END_IF;
IF r8_to_r10 AND r8.fire AND r10.insert_reset THEN r8.fire := FALSE; END_IF;

(* Network 48 *)
Easy_Sort_2_reset:
IF r8.reset THEN r8.fire := FALSE; END_IF;

(* Network 49 *)
Easy_Sort_3_clear_dest:
_e17(CLK := r9.fire);
IF _e17.Q THEN r9.destination := 0; END_IF;

(* Network 50 *)
Easy_Sort_3_lockout:
r9.lockout := r7.fire OR r8.fire OR r9.fire OR r21.fire;

(* Network 51 *)
Easy_Sort_3_io_ok:
r9.waiting := NOT r9.lockout AND NOT r9.custom_send_lock AND r9.front AND r9.done;

(* Network 52 *)
Easy_Sort_3_to_r10_P1:
r9_to_r10 := r9.destination = 10;

(* Network 53 *)
Easy_Sort_3_to_r10_P2:
_p18 := r9_to_r10 AND NOT r10.going_to AND NOT r9.reset AND NOT r10.insert_reset;
IF _p18 THEN
    r10.going_to := TRUE;
    r9.fire := TRUE;
END_IF;
IF r9_to_r10 AND r9.fire AND r10.insert_reset THEN r9.fire := FALSE; END_IF;

(* Network 54 *)
Easy_Sort_3_reset:
IF r9.reset THEN r9.fire := FALSE; END_IF;

(* Network 55 *)
Transfer_Rail_clear_dest:
_e19(CLK := r10.fire);
IF _e19.Q THEN r10.destination := 0; END_IF;

(* Network 56 *)
Transfer_Rail_lockout:
r10.lockout := r10.fire;

(* Network 57 *)
Transfer_Rail_io_ok:
r10.waiting := NOT r10.lockout AND NOT r10.custom_send_lock AND r10.front AND r10.down AND r10.fire_down AND NOT r10.up AND NOT r10.fire_up AND NOT r10.after;

(* Network 58 *)
Transfer_Rail_to_r11_P1:
r10_to_r11 := r10.destination = 11;

(* Network 59 *)
Transfer_Rail_to_r11_P2:
_p20 := r10_to_r11 AND NOT r11.going_to AND NOT r10.reset AND NOT r11.insert_reset;
IF _p20 THEN
    r11.going_to := TRUE;
    r10.fire := TRUE;
END_IF;
IF r10_to_r11 AND r10.fire AND r11.insert_reset THEN r10.fire := FALSE; END_IF;

(* Network 60 *)
Transfer_Rail_reset:
IF r10.reset THEN r10.fire := FALSE; END_IF;

(* Network 61 *)
Pre_Storage_1_clear_dest:
_e21(CLK := r11.fire);
IF _e21.Q THEN r11.destination := 0; END_IF;

(* Network 62 *)
Pre_Storage_1_lockout:
r11.lockout := r11.fire;

(* Network 63 *)
Pre_Storage_1_io_ok:
r11.waiting := NOT r11.lockout AND NOT r11.custom_send_lock AND r11.front AND NOT r11.after;

(* Network 64 *)
Pre_Storage_1_to_r12_P1:
r11_to_r12 := r11.destination = 12;

(* Network 65 *)
Pre_Storage_1_to_r12_P2:
_p22 := r11_to_r12 AND NOT r12.going_to AND NOT r11.reset AND NOT r12.insert_reset;
IF _p22 THEN
    r12.going_to := TRUE;
    r11.fire := TRUE;
END_IF;
IF r11_to_r12 AND r11.fire AND r12.insert_reset THEN r11.fire := FALSE; END_IF;

(* Network 66 *)
Pre_Storage_1_reset:
IF r11.reset THEN r11.fire := FALSE; END_IF;

(* Network 67 *)
Pre_Storage_2_clear_dest:
_e23(CLK := r12.fire);
IF _e23.Q THEN r12.destination := 0; END_IF;

(* Network 68 *)
Pre_Storage_2_lockout:
r12.lockout := r12.fire;

(* Network 69 *)
Pre_Storage_2_io_ok:
r12.waiting := NOT r12.lockout AND NOT r12.custom_send_lock AND r12.front AND NOT r12.after;

(* Network 70 *)
Pre_Storage_2_to_r13_P1:
r12_to_r13 := r12.destination = 13;

(* Network 71 *)
Pre_Storage_2_to_r13_P2:
_p24 := r12_to_r13 AND NOT r13.going_to AND NOT r12.reset AND NOT r13.insert_reset;
IF _p24 THEN
    r13.going_to := TRUE;
    r12.fire := TRUE;
END_IF;
IF r12_to_r13 AND r12.fire AND r13.insert_reset THEN r12.fire := FALSE; END_IF;

(* Network 72 *)
Pre_Storage_2_reset:
IF r12.reset THEN r12.fire := FALSE; END_IF;

(* Network 73 *)
Belt_Opener_Rail_clear_dest:
_e25(CLK := r13.fire);
IF _e25.Q THEN r13.destination := 0; END_IF;

(* Network 74 *)
Belt_Opener_Rail_lockout:
r13.lockout := r13.fire;

(* Network 75 *)
Belt_Opener_Rail_io_ok:
r13.waiting := NOT r13.lockout AND NOT r13.custom_send_lock AND r13.front AND r13.done AND NOT r13.after;

(* Network 76 *)
Belt_Opener_Rail_to_r14_P1:
r13_to_r14 := r13.destination = 14;

(* Network 77 *)
Belt_Opener_Rail_to_r14_P2:
_p26 := r13_to_r14 AND NOT r14.going_to AND NOT r13.reset AND NOT r14.insert_reset;
IF _p26 THEN
    r14.going_to := TRUE;
    r13.fire := TRUE;
END_IF;
IF r13_to_r14 AND r13.fire AND r14.insert_reset THEN r13.fire := FALSE; END_IF;

(* Network 78 *)
Belt_Opener_Rail_to_r15_P1:
r13_to_r15 := r13.destination = 15;

(* Network 79 *)
Belt_Opener_Rail_to_r15_P2:
_p27 := r13_to_r15 AND NOT r15.going_to AND NOT r13.reset AND NOT r15.insert_reset;
IF _p27 THEN
    r15.going_to := TRUE;
    r13.fire := TRUE;
END_IF;
IF r13_to_r15 AND r13.fire AND r15.insert_reset THEN r13.fire := FALSE; END_IF;

(* Network 80 *)
Belt_Opener_Rail_to_r16_P1:
r13_to_r16 := r13.destination = 16;

(* Network 81 *)
Belt_Opener_Rail_to_r16_P2:
_p28 := r13_to_r16 AND NOT r16.going_to AND NOT r13.reset AND NOT r16.insert_reset;
IF _p28 THEN
    r16.going_to := TRUE;
    r13.fire := TRUE;
END_IF;
IF r13_to_r16 AND r13.fire AND r16.insert_reset THEN r13.fire := FALSE; END_IF;

(* Network 82 *)
Belt_Opener_Rail_reset:
IF r13.reset THEN r13.fire := FALSE; END_IF;

(* Network 83 *)
Storage_Rail_1_clear_dest:
_e29(CLK := r14.fire);
IF _e29.Q THEN r14.destination := 0; END_IF;

(* Network 84 *)
Storage_Rail_1_lockout:
r14.lockout := r14.fire OR r15.fire OR r18.fire;

(* Network 85 *)
Storage_Rail_1_io_ok:
r14.waiting := NOT r14.lockout AND NOT r14.custom_send_lock AND r14.front AND NOT r14.after;

(* Network 86 *)
Storage_Rail_1_to_r19_P1:
r14_to_r19 := r14.destination = 19;

(* Network 87 *)
Storage_Rail_1_to_r19_P2:
_p30 := r14_to_r19 AND NOT r19.going_to AND NOT r14.reset AND NOT r19.insert_reset;
IF _p30 THEN
    r19.going_to := TRUE;
    r14.fire := TRUE;
END_IF;
IF r14_to_r19 AND r14.fire AND r19.insert_reset THEN r14.fire := FALSE; END_IF;

(* Network 88 *)
Storage_Rail_1_reset:
IF r14.reset THEN r14.fire := FALSE; END_IF;

(* Network 89 *)
Storage_Rail_2_clear_dest:
_e31(CLK := r15.fire);
IF _e31.Q THEN r15.destination := 0; END_IF;

(* Network 90 *)
Storage_Rail_2_lockout:
r15.lockout := r14.fire OR r15.fire OR r18.fire;

(* Network 91 *)
Storage_Rail_2_io_ok:
r15.waiting := NOT r15.lockout AND NOT r15.custom_send_lock AND r15.front AND NOT r15.after;

(* Network 92 *)
Storage_Rail_2_to_r19_P1:
r15_to_r19 := r15.destination = 19;

(* Network 93 *)
Storage_Rail_2_to_r19_P2:
_p32 := r15_to_r19 AND NOT r19.going_to AND NOT r15.reset AND NOT r19.insert_reset;
IF _p32 THEN
    r19.going_to := TRUE;
    r15.fire := TRUE;
END_IF;
IF r15_to_r19 AND r15.fire AND r19.insert_reset THEN r15.fire := FALSE; END_IF;

(* Network 94 *)
Storage_Rail_2_reset:
IF r15.reset THEN r15.fire := FALSE; END_IF;

(* Network 95 *)
Storage_Rail_3_clear_dest:
_e33(CLK := r16.fire);
IF _e33.Q THEN r16.destination := 0; END_IF;

(* Network 96 *)
Storage_Rail_3_lockout:
r16.lockout := r16.fire;

(* Network 97 *)
Storage_Rail_3_io_ok:
r16.waiting := NOT r16.lockout AND NOT r16.custom_send_lock AND r16.front AND NOT r16.after;

(* Network 98 *)
Storage_Rail_3_to_r17_P1:
r16_to_r17 := r16.destination = 17;

(* Network 99 *)
Storage_Rail_3_to_r17_P2:
_p34 := r16_to_r17 AND NOT r17.going_to AND NOT r16.reset AND NOT r17.insert_reset;
IF _p34 THEN
    r17.going_to := TRUE;
    r16.fire := TRUE;
END_IF;
IF r16_to_r17 AND r16.fire AND r17.insert_reset THEN r16.fire := FALSE; END_IF;

(* Network 100 *)
Storage_Rail_3_reset:
IF r16.reset THEN r16.fire := FALSE; END_IF;

(* Network 101 *)
Storage_Opener_clear_dest:
_e35(CLK := r17.fire);
IF _e35.Q THEN r17.destination := 0; END_IF;

(* Network 102 *)
Storage_Opener_lockout:
r17.lockout := r17.fire;

(* Network 103 *)
Storage_Opener_io_ok:
r17.waiting := NOT r17.lockout AND NOT r17.custom_send_lock AND r17.front AND r17.done AND NOT r17.after;

(* Network 104 *)
Storage_Opener_to_r18_P1:
r17_to_r18 := r17.destination = 18;

(* Network 105 *)
Storage_Opener_to_r18_P2:
_p36 := r17_to_r18 AND NOT r18.going_to AND NOT r17.reset AND NOT r18.insert_reset;
IF _p36 THEN
    r18.going_to := TRUE;
    r17.fire := TRUE;
END_IF;
IF r17_to_r18 AND r17.fire AND r18.insert_reset THEN r17.fire := FALSE; END_IF;

(* Network 106 *)
Storage_Opener_reset:
IF r17.reset THEN r17.fire := FALSE; END_IF;

(* Network 107 *)
Empty_1_clear_dest:
_e37(CLK := r18.fire);
IF _e37.Q THEN r18.destination := 0; END_IF;

(* Network 108 *)
Empty_1_lockout:
r18.lockout := r14.fire OR r15.fire OR r18.fire;

(* Network 109 *)
Empty_1_io_ok:
r18.waiting := NOT r18.lockout AND NOT r18.custom_send_lock AND r18.front AND NOT r18.after;

(* Network 110 *)
Empty_1_to_r19_P1:
r18_to_r19 := r18.destination = 19;

(* Network 111 *)
Empty_1_to_r19_P2:
_p38 := r18_to_r19 AND NOT r19.going_to AND NOT r18.reset AND NOT r19.insert_reset;
IF _p38 THEN
    r19.going_to := TRUE;
    r18.fire := TRUE;
END_IF;
IF r18_to_r19 AND r18.fire AND r19.insert_reset THEN r18.fire := FALSE; END_IF;

(* Network 112 *)
Empty_1_reset:
IF r18.reset THEN r18.fire := FALSE; END_IF;

(* Network 113 *)
Empty_2_clear_dest:
_e39(CLK := r19.fire);
IF _e39.Q THEN r19.destination := 0; END_IF;

(* Network 114 *)
Empty_2_lockout:
r19.lockout := r19.fire;

(* Network 115 *)
Empty_2_io_ok:
r19.waiting := NOT r19.lockout AND NOT r19.custom_send_lock AND r19.front AND NOT r19.after;

(* Network 116 *)
Empty_2_to_r20_P1:
r19_to_r20 := r19.destination = 20;

(* Network 117 *)
Empty_2_to_r20_P2:
_p40 := r19_to_r20 AND NOT r20.going_to AND NOT r19.reset AND NOT r20.insert_reset;
IF _p40 THEN
    r20.going_to := TRUE;
    r19.fire := TRUE;
END_IF;
IF r19_to_r20 AND r19.fire AND r20.insert_reset THEN r19.fire := FALSE; END_IF;

(* Network 118 *)
Empty_2_reset:
IF r19.reset THEN r19.fire := FALSE; END_IF;

(* Network 119 *)
Empty_3_Lift_clear_dest:
_e41(CLK := r20.fire);
IF _e41.Q THEN r20.destination := 0; END_IF;

(* Network 120 *)
Empty_3_Lift_lockout:
r20.lockout := r20.fire;

(* Network 121 *)
Empty_3_Lift_io_ok:
r20.waiting := NOT r20.lockout AND NOT r20.custom_send_lock AND r20.front AND r20.up AND r20.fire_up AND NOT r20.down AND NOT r20.fire_down AND NOT r20.after;

(* Network 122 *)
Empty_3_Lift_to_r21_P1:
r20_to_r21 := r20.destination = 21;

(* Network 123 *)
Empty_3_Lift_to_r21_P2:
_p42 := r20_to_r21 AND NOT r21.going_to AND NOT r20.reset AND NOT r21.insert_reset;
IF _p42 THEN
    r21.going_to := TRUE;
    r20.fire := TRUE;
END_IF;
IF r20_to_r21 AND r20.fire AND r21.insert_reset THEN r20.fire := FALSE; END_IF;

(* Network 124 *)
Empty_3_Lift_reset:
IF r20.reset THEN r20.fire := FALSE; END_IF;

(* Network 125 *)
Empty_4_clear_dest:
_e43(CLK := r21.fire);
IF _e43.Q THEN r21.destination := 0; END_IF;

(* Network 126 *)
Empty_4_lockout:
r21.lockout := r7.fire OR r8.fire OR r9.fire OR r21.fire;

(* Network 127 *)
Empty_4_io_ok:
r21.waiting := NOT r21.lockout AND NOT r21.custom_send_lock AND r21.front AND NOT r21.after;

(* Network 128 *)
Empty_4_to_r10_P1:
r21_to_r10 := r21.destination = 10;

(* Network 129 *)
Empty_4_to_r10_P2:
_p44 := r21_to_r10 AND NOT r10.going_to AND NOT r21.reset AND NOT r10.insert_reset;
IF _p44 THEN
    r10.going_to := TRUE;
    r21.fire := TRUE;
END_IF;
IF r21_to_r10 AND r21.fire AND r10.insert_reset THEN r21.fire := FALSE; END_IF;

(* Network 130 *)
Empty_4_reset:
IF r21.reset THEN r21.fire := FALSE; END_IF;
END_PROGRAM
```

### Program Logical/OPENERS (IEC, version 1.00.1)

#### OPENERS.st
```iecst
(********************************************************************
 * Program: openers
 * File: openers.st
 ********************************************************************)
PROGRAM _CYCLIC
END_PROGRAM
```

### Program Logical/CLOSERS (IEC, version 1.00.1)

#### CLOSERS.st
```iecst
(********************************************************************
 * Program: closers
 * File: closers.st
 ********************************************************************)
PROGRAM _CYCLIC
END_PROGRAM
```

### Program Logical/SWITCHES (IEC, version 1.00.1)

#### SWITCHES.st
```iecst
(********************************************************************
 * Program: switches
 * File: switches.st
 ********************************************************************)
PROGRAM _CYCLIC
END_PROGRAM
```

#### Cyclic.ld - not listed in the package file held
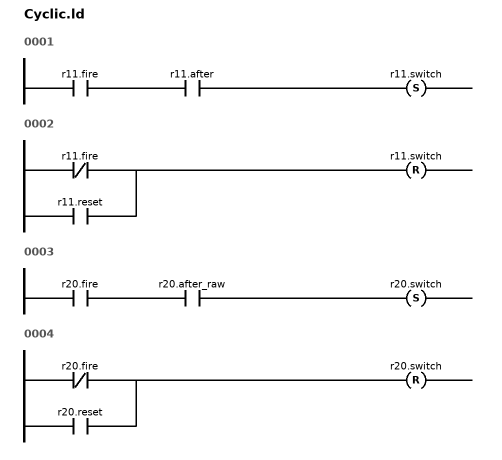
Ladder, written as Structured Text:
```iecst
PROGRAM _CYCLIC
(* Network 1 *)
IF r11.fire AND r11.after THEN r11.switch := TRUE; END_IF;

(* Network 2 *)
IF NOT r11.fire OR r11.reset THEN r11.switch := FALSE; END_IF;

(* Network 3 *)
IF r20.fire AND r20.after_raw THEN r20.switch := TRUE; END_IF;

(* Network 4 *)
IF NOT r20.fire OR r20.reset THEN r20.switch := FALSE; END_IF;
END_PROGRAM
```

### Program Logical/IO_SCANNING (IEC, version 1.00.1) - IO_SCANNING

#### IO_SCANNING.st
```iecst
(********************************************************************
 * Program: io_scanning
 * File: io_scanning.st
 ********************************************************************)
PROGRAM _INIT
  (* --------------------------------------------------------------------
  Reset FUNCTION blocks AND data structure on startup (SGC)
  --------------------------------------------------------------------- *)

END_PROGRAM
```

### Program Logical/SORTS (IEC, version 1.00.1) - SORTS

#### SORTS.st
```iecst
(********************************************************************
 * Program: sorts
 * File: sorts.st
 ********************************************************************)
PROGRAM _CYCLIC

END_PROGRAM
```

### Program Logical/WARNINGS (IEC, version 1.00.1) - WARNINGS

#### WARNINGS.st
```iecst
(********************************************************************
 * Program: warnings
 * File: warnings.st
 ********************************************************************)
PROGRAM _CYCLIC
END_PROGRAM
```

### Program Logical/TRANSFERS (IEC, version 1.00.1) - TRANSFERS

#### TRANSFERS.st
```iecst
(********************************************************************
 * Program: transfers
 * File: transfers.st
 ********************************************************************)
PROGRAM _CYCLIC
END_PROGRAM
```

### Program Logical/custom (IEC)
